gfCNCPoint5[19231] = {X 227.6405, Y 45.0000, Z -7.1667, A 0.000, B 0.000, C 0.000 }
gfCNCPoint5[19232] = {X 227.5362, Y 45.9257, Z -7.1667, A 0.000, B 0.000, C 0.000 }
gfCNCPoint5[19233] = {X 227.2285, Y 46.8050, Z -7.1667, A 0.000, B 0.000, C 0.000 }
gfCNCPoint5[19234] = {X 226.7329, Y 47.5937, Z -7.1667, A 0.000, B 0.000, C 0.000 }
gfCNCPoint5[19235] = {X 226.0742, Y 48.2524, Z -7.1667, A 0.000, B 0.000, C 0.000 }
gfCNCPoint5[19236] = {X 225.2854, Y 48.7480, Z -7.1667, A 0.000, B 0.000, C 0.000 }
gfCNCPoint5[19237] = {X 224.4062, Y 49.0557, Z -7.1667, A 0.000, B 0.000, C 0.000 }
gfCNCPoint5[19238] = {X 223.4805, Y 49.1600, Z -7.1667, A 0.000, B 0.000, C 0.000 }
gfCNCPoint5[19239] = {X 217.0370, Y 49.1600, Z -7.1667, A 0.000, B 0.000, C 0.000 }
gfCNCPoint5[19240] = {X 216.1160, Y 49.0568, Z -7.1667, A 0.000, B 0.000, C 0.000 }
gfCNCPoint5[19241] = {X 215.2406, Y 48.7521, Z -7.1667, A 0.000, B 0.000, C 0.000 }
gfCNCPoint5[19242] = {X 214.4544, Y 48.2613, Z -7.1667, A 0.000, B 0.000, C 0.000 }
gfCNCPoint5[19243] = {X 213.7965, Y 47.6085, Z -7.1667, A 0.000, B 0.000, C 0.000 }
gfCNCPoint5[19244] = {X 213.2993, Y 46.8263, Z -7.1667, A 0.000, B 0.000, C 0.000 }
gfCNCPoint5[19245] = {X 212.9877, Y 45.9534, Z -7.1667, A 0.000, B 0.000, C 0.000 }
gfCNCPoint5[19246] = {X 212.8771, Y 45.0332, Z -7.1667, A 0.000, B 0.000, C 0.000 }
gfCNCPoint5[19247] = {X 212.8770, Y 44.1909, Z -7.1667, A 0.000, B 0.000, C 0.000 }
gfCNCPoint5[19248] = {X 212.9460, Y 43.4438, Z -7.1667, A 0.000, B 0.000, C 0.000 }
gfCNCPoint5[19249] = {X 213.1506, Y 42.7220, Z -7.1667, A 0.000, B 0.000, C 0.000 }
gfCNCPoint5[19250] = {X 213.4838, Y 42.0498, Z -7.1667, A 0.000, B 0.000, C 0.000 }
gfCNCPoint5[19251] = {X 213.9345, Y 41.4500, Z -7.1667, A 0.000, B 0.000, C 0.000 }
gfCNCPoint5[19252] = {X 214.3990, Y 40.9376, Z -7.1667, A 0.000, B 0.000, C 0.000 }
gfCNCPoint5[19253] = {X 214.4039, Y 40.3069, Z -7.1667, A 0.000, B 0.000, C 0.000 }
gfCNCPoint5[19254] = {X 214.4039, Y 28.5737, Z -7.1667, A 0.000, B 0.000, C 0.000 }
gfCNCPoint5[19255] = {X 210.4039, Y 28.5737, Z -7.1667, A 0.000, B 0.000, C 0.000 }
gfCNCPoint5[19256] = {X 214.4839, Y 28.5737, Z -7.1667, A 0.000, B 0.000, C 0.000 }
gfCNCPoint5[19257] = {X 214.4839, Y 17.4614, Z -7.1667, A 0.000, B 0.000, C 0.000 }
gfCNCPoint5[19258] = {X 214.4785, Y 16.7691, Z -7.1667, A 0.000, B 0.000, C 0.000 }
gfCNCPoint5[19259] = {X 214.4828, Y 16.1596, Z -7.1667, A 0.000, B 0.000, C 0.000 }
gfCNCPoint5[19260] = {X 214.4247, Y 16.1121, Z -7.1667, A 0.000, B 0.000, C 0.000 }
gfCNCPoint5[19261] = {X 214.3675, Y 16.0635, Z -7.1667, A 0.000, B 0.000, C 0.000 }
gfCNCPoint5[19262] = {X 213.7773, Y 15.4317, Z -7.1667, A 0.000, B 0.000, C 0.000 }
gfCNCPoint5[19263] = {X 213.3335, Y 14.6898, Z -7.1667, A 0.000, B 0.000, C 0.000 }
gfCNCPoint5[19264] = {X 213.0559, Y 13.8710, Z -7.1667, A 0.000, B 0.000, C 0.000 }
gfCNCPoint5[19265] = {X 212.9572, Y 13.0121, Z -7.1667, A 0.000, B 0.000, C 0.000 }
gfCNCPoint5[19266] = {X 212.9570, Y 12.1868, Z -7.1667, A 0.000, B 0.000, C 0.000 }
gfCNCPoint5[19267] = {X 213.0593, Y 11.2789, Z -7.1667, A 0.000, B 0.000, C 0.000 }
gfCNCPoint5[19268] = {X 213.3611, Y 10.4166, Z -7.1667, A 0.000, B 0.000, C 0.000 }
gfCNCPoint5[19269] = {X 213.8471, Y 9.6430, Z -7.1667, A 0.000, B 0.000, C 0.000 }
gfCNCPoint5[19270] = {X 214.4932, Y 8.9969, Z -7.1667, A 0.000, B 0.000, C 0.000 }
gfCNCPoint5[19271] = {X 215.2668, Y 8.5109, Z -7.1667, A 0.000, B 0.000, C 0.000 }
gfCNCPoint5[19272] = {X 216.1291, Y 8.2091, Z -7.1667, A 0.000, B 0.000, C 0.000 }
gfCNCPoint5[19273] = {X 217.0370, Y 8.1068, Z -7.1667, A 0.000, B 0.000, C 0.000 }
gfCNCPoint5[19274] = {X 223.4805, Y 8.1068, Z -7.1667, A 0.000, B 0.000, C 0.000 }
gfCNCPoint5[19275] = {X 224.3884, Y 8.2091, Z -7.1667, A 0.000, B 0.000, C 0.000 }
gfCNCPoint5[19276] = {X 225.2507, Y 8.5109, Z -7.1667, A 0.000, B 0.000, C 0.000 }
gfCNCPoint5[19277] = {X 226.0243, Y 8.9969, Z -7.1667, A 0.000, B 0.000, C 0.000 }
gfCNCPoint5[19278] = {X 226.6704, Y 9.6430, Z -7.1667, A 0.000, B 0.000, C 0.000 }
gfCNCPoint5[19279] = {X 227.1564, Y 10.4166, Z -7.1667, A 0.000, B 0.000, C 0.000 }
gfCNCPoint5[19280] = {X 227.4582, Y 11.2789, Z -7.1667, A 0.000, B 0.000, C 0.000 }
gfCNCPoint5[19281] = {X 227.5605, Y 12.1868, Z -7.1667, A 0.000, B 0.000, C 0.000 }
gfCNCPoint5[19282] = {X 227.5605, Y 12.9782, Z -7.1667, A 0.000, B 0.000, C 0.000 }
gfCNCPoint5[19283] = {X 227.4589, Y 13.8829, Z -7.1667, A 0.000, B 0.000, C 0.000 }
gfCNCPoint5[19284] = {X 227.1591, Y 14.7427, Z -7.1667, A 0.000, B 0.000, C 0.000 }
gfCNCPoint5[19285] = {X 226.6762, Y 15.5145, Z -7.1667, A 0.000, B 0.000, C 0.000 }
gfCNCPoint5[19286] = {X 226.0341, Y 16.1600, Z -7.1667, A 0.000, B 0.000, C 0.000 }
gfCNCPoint5[19287] = {X 226.0351, Y 41.0283, Z -7.1667, A 0.000, B 0.000, C 0.000 }
gfCNCPoint5[19288] = {X 226.1412, Y 41.1157, Z -7.1667, A 0.000, B 0.000, C 0.000 }
gfCNCPoint5[19289] = {X 226.7344, Y 41.7474, Z -7.1667, A 0.000, B 0.000, C 0.000 }
gfCNCPoint5[19290] = {X 227.1808, Y 42.4901, Z -7.1667, A 0.000, B 0.000, C 0.000 }
gfCNCPoint5[19291] = {X 227.4603, Y 43.3104, Z -7.1667, A 0.000, B 0.000, C 0.000 }
gfCNCPoint5[19292] = {X 227.5603, Y 44.1712, Z -7.1667, A 0.000, B 0.000, C 0.000 }
gfCNCPoint5[19293] = {X 227.5605, Y 45.0000, Z -7.1667, A 0.000, B 0.000, C 0.000 }
gfCNCPoint5[19294] = {X 227.4582, Y 45.9079, Z -7.1667, A 0.000, B 0.000, C 0.000 }
gfCNCPoint5[19295] = {X 227.1564, Y 46.7702, Z -7.1667, A 0.000, B 0.000, C 0.000 }
gfCNCPoint5[19296] = {X 226.6704, Y 47.5438, Z -7.1667, A 0.000, B 0.000, C 0.000 }
gfCNCPoint5[19297] = {X 226.0243, Y 48.1899, Z -7.1667, A 0.000, B 0.000, C 0.000 }
gfCNCPoint5[19298] = {X 225.2507, Y 48.6760, Z -7.1667, A 0.000, B 0.000, C 0.000 }
gfCNCPoint5[19299] = {X 224.3884, Y 48.9777, Z -7.1667, A 0.000, B 0.000, C 0.000 }
gfCNCPoint5[19300] = {X 223.4805, Y 49.0800, Z -7.1667, A 0.000, B 0.000, C 0.000 }
gfCNCPoint5[19301] = {X 217.0370, Y 49.0800, Z -7.1667, A 0.000, B 0.000, C 0.000 }
gfCNCPoint5[19302] = {X 216.1337, Y 48.9787, Z -7.1667, A 0.000, B 0.000, C 0.000 }
gfCNCPoint5[19303] = {X 215.2752, Y 48.6800, Z -7.1667, A 0.000, B 0.000, C 0.000 }
gfCNCPoint5[19304] = {X 214.5041, Y 48.1986, Z -7.1667, A 0.000, B 0.000, C 0.000 }
gfCNCPoint5[19305] = {X 213.8588, Y 47.5584, Z -7.1667, A 0.000, B 0.000, C 0.000 }
gfCNCPoint5[19306] = {X 213.3712, Y 46.7912, Z -7.1667, A 0.000, B 0.000, C 0.000 }
gfCNCPoint5[19307] = {X 213.0656, Y 45.9351, Z -7.1667, A 0.000, B 0.000, C 0.000 }
gfCNCPoint5[19308] = {X 212.9571, Y 45.0325, Z -7.1667, A 0.000, B 0.000, C 0.000 }
gfCNCPoint5[19309] = {X 212.9570, Y 44.1909, Z -7.1667, A 0.000, B 0.000, C 0.000 }
gfCNCPoint5[19310] = {X 213.0246, Y 43.4585, Z -7.1667, A 0.000, B 0.000, C 0.000 }
gfCNCPoint5[19311] = {X 213.2252, Y 42.7508, Z -7.1667, A 0.000, B 0.000, C 0.000 }
gfCNCPoint5[19312] = {X 213.5519, Y 42.0918, Z -7.1667, A 0.000, B 0.000, C 0.000 }
gfCNCPoint5[19313] = {X 213.9938, Y 41.5037, Z -7.1667, A 0.000, B 0.000, C 0.000 }
gfCNCPoint5[19314] = {X 214.4788, Y 40.9687, Z -7.1667, A 0.000, B 0.000, C 0.000 }
gfCNCPoint5[19315] = {X 214.4839, Y 40.3072, Z -7.1667, A 0.000, B 0.000, C 0.000 }
gfCNCPoint5[19316] = {X 214.4839, Y 28.5737, Z -7.1667, A 0.000, B 0.000, C 0.000 }
gfCNCPoint5[19317] = {X 210.4839, Y 28.5737, Z -7.1667, A 0.000, B 0.000, C 0.000 }
gfCNCPoint5[19318] = {X 214.5639, Y 28.5737, Z -7.1667, A 0.000, B 0.000, C 0.000 }
gfCNCPoint5[19319] = {X 214.5639, Y 17.4611, Z -7.1667, A 0.000, B 0.000, C 0.000 }
gfCNCPoint5[19320] = {X 214.5585, Y 16.7687, Z -7.1667, A 0.000, B 0.000, C 0.000 }
gfCNCPoint5[19321] = {X 214.5580, Y 16.1871, Z -7.1667, A 0.000, B 0.000, C 0.000 }
gfCNCPoint5[19322] = {X 214.5756, Y 16.1310, Z -7.1667, A 0.000, B 0.000, C 0.000 }
gfCNCPoint5[19323] = {X 214.4969, Y 16.0680, Z -7.1667, A 0.000, B 0.000, C 0.000 }
gfCNCPoint5[19324] = {X 214.4199, Y 16.0030, Z -7.1667, A 0.000, B 0.000, C 0.000 }
gfCNCPoint5[19325] = {X 213.8362, Y 15.3769, Z -7.1667, A 0.000, B 0.000, C 0.000 }
gfCNCPoint5[19326] = {X 213.3991, Y 14.6410, Z -7.1667, A 0.000, B 0.000, C 0.000 }
gfCNCPoint5[19327] = {X 213.1286, Y 13.8290, Z -7.1667, A 0.000, B 0.000, C 0.000 }
gfCNCPoint5[19328] = {X 213.0370, Y 12.9780, Z -7.1667, A 0.000, B 0.000, C 0.000 }
gfCNCPoint5[19329] = {X 213.0370, Y 12.1868, Z -7.1667, A 0.000, B 0.000, C 0.000 }
gfCNCPoint5[19330] = {X 213.1373, Y 11.2967, Z -7.1667, A 0.000, B 0.000, C 0.000 }
gfCNCPoint5[19331] = {X 213.4331, Y 10.4513, Z -7.1667, A 0.000, B 0.000, C 0.000 }
gfCNCPoint5[19332] = {X 213.9097, Y 9.6929, Z -7.1667, A 0.000, B 0.000, C 0.000 }
gfCNCPoint5[19333] = {X 214.5431, Y 9.0595, Z -7.1667, A 0.000, B 0.000, C 0.000 }
gfCNCPoint5[19334] = {X 215.3015, Y 8.5829, Z -7.1667, A 0.000, B 0.000, C 0.000 }
gfCNCPoint5[19335] = {X 216.1469, Y 8.2871, Z -7.1667, A 0.000, B 0.000, C 0.000 }
gfCNCPoint5[19336] = {X 217.0370, Y 8.1868, Z -7.1667, A 0.000, B 0.000, C 0.000 }
gfCNCPoint5[19337] = {X 223.4805, Y 8.1868, Z -7.1667, A 0.000, B 0.000, C 0.000 }
gfCNCPoint5[19338] = {X 224.3706, Y 8.2871, Z -7.1667, A 0.000, B 0.000, C 0.000 }
gfCNCPoint5[19339] = {X 225.2160, Y 8.5829, Z -7.1667, A 0.000, B 0.000, C 0.000 }
gfCNCPoint5[19340] = {X 225.9744, Y 9.0595, Z -7.1667, A 0.000, B 0.000, C 0.000 }
gfCNCPoint5[19341] = {X 226.6078, Y 9.6929, Z -7.1667, A 0.000, B 0.000, C 0.000 }
gfCNCPoint5[19342] = {X 227.0844, Y 10.4513, Z -7.1667, A 0.000, B 0.000, C 0.000 }
gfCNCPoint5[19343] = {X 227.3802, Y 11.2967, Z -7.1667, A 0.000, B 0.000, C 0.000 }
gfCNCPoint5[19344] = {X 227.4805, Y 12.1868, Z -7.1667, A 0.000, B 0.000, C 0.000 }
gfCNCPoint5[19345] = {X 227.4803, Y 13.0192, Z -7.1667, A 0.000, B 0.000, C 0.000 }
gfCNCPoint5[19346] = {X 227.3717, Y 13.9045, Z -7.1667, A 0.000, B 0.000, C 0.000 }
gfCNCPoint5[19347] = {X 227.0697, Y 14.7437, Z -7.1667, A 0.000, B 0.000, C 0.000 }
gfCNCPoint5[19348] = {X 226.5892, Y 15.4951, Z -7.1667, A 0.000, B 0.000, C 0.000 }
gfCNCPoint5[19349] = {X 225.9541, Y 16.1214, Z -7.1667, A 0.000, B 0.000, C 0.000 }
gfCNCPoint5[19350] = {X 225.9551, Y 41.0660, Z -7.1667, A 0.000, B 0.000, C 0.000 }
gfCNCPoint5[19351] = {X 226.0938, Y 41.1805, Z -7.1667, A 0.000, B 0.000, C 0.000 }
gfCNCPoint5[19352] = {X 226.6790, Y 41.8068, Z -7.1667, A 0.000, B 0.000, C 0.000 }
gfCNCPoint5[19353] = {X 227.1173, Y 42.5435, Z -7.1667, A 0.000, B 0.000, C 0.000 }
gfCNCPoint5[19354] = {X 227.3886, Y 43.3566, Z -7.1667, A 0.000, B 0.000, C 0.000 }
gfCNCPoint5[19355] = {X 227.4805, Y 44.2089, Z -7.1667, A 0.000, B 0.000, C 0.000 }
gfCNCPoint5[19356] = {X 227.4805, Y 45.0000, Z -7.1667, A 0.000, B 0.000, C 0.000 }
gfCNCPoint5[19357] = {X 227.3802, Y 45.8901, Z -7.1667, A 0.000, B 0.000, C 0.000 }
gfCNCPoint5[19358] = {X 227.0844, Y 46.7355, Z -7.1667, A 0.000, B 0.000, C 0.000 }
gfCNCPoint5[19359] = {X 226.6078, Y 47.4940, Z -7.1667, A 0.000, B 0.000, C 0.000 }
gfCNCPoint5[19360] = {X 225.9744, Y 48.1273, Z -7.1667, A 0.000, B 0.000, C 0.000 }
gfCNCPoint5[19361] = {X 225.2160, Y 48.6039, Z -7.1667, A 0.000, B 0.000, C 0.000 }
gfCNCPoint5[19362] = {X 224.3706, Y 48.8997, Z -7.1667, A 0.000, B 0.000, C 0.000 }
gfCNCPoint5[19363] = {X 223.4805, Y 49.0000, Z -7.1667, A 0.000, B 0.000, C 0.000 }
gfCNCPoint5[19364] = {X 217.0370, Y 49.0000, Z -7.1667, A 0.000, B 0.000, C 0.000 }
gfCNCPoint5[19365] = {X 216.1469, Y 48.8997, Z -7.1667, A 0.000, B 0.000, C 0.000 }
gfCNCPoint5[19366] = {X 215.3015, Y 48.6039, Z -7.1667, A 0.000, B 0.000, C 0.000 }
gfCNCPoint5[19367] = {X 214.5430, Y 48.1273, Z -7.1667, A 0.000, B 0.000, C 0.000 }
gfCNCPoint5[19368] = {X 213.9097, Y 47.4939, Z -7.1667, A 0.000, B 0.000, C 0.000 }
gfCNCPoint5[19369] = {X 213.4331, Y 46.7355, Z -7.1667, A 0.000, B 0.000, C 0.000 }
gfCNCPoint5[19370] = {X 213.1373, Y 45.8901, Z -7.1667, A 0.000, B 0.000, C 0.000 }
gfCNCPoint5[19371] = {X 213.0370, Y 45.0000, Z -7.1667, A 0.000, B 0.000, C 0.000 }
gfCNCPoint5[19372] = {X 213.0370, Y 44.1909, Z -7.1667, A 0.000, B 0.000, C 0.000 }
gfCNCPoint5[19373] = {X 213.1546, Y 43.2380, Z -7.1667, A 0.000, B 0.000, C 0.000 }
gfCNCPoint5[19374] = {X 213.5002, Y 42.3423, Z -7.1667, A 0.000, B 0.000, C 0.000 }
gfCNCPoint5[19375] = {X 214.0531, Y 41.5574, Z -7.1667, A 0.000, B 0.000, C 0.000 }
gfCNCPoint5[19376] = {X 214.5585, Y 40.9999, Z -7.1667, A 0.000, B 0.000, C 0.000 }
gfCNCPoint5[19377] = {X 214.5639, Y 40.3075, Z -7.1667, A 0.000, B 0.000, C 0.000 }
gfCNCPoint5[19378] = {X 214.5639, Y 28.5737, Z -7.1667, A 0.000, B 0.000, C 0.000 }
gfCNCPoint5[19379] = {X 210.4839, Y 28.5737, Z -7.1667, A 0.000, B 0.000, C 0.000 }
gfCNCPoint5[19380] = {X 210.4839, Y 28.5737, Z -4.1667, A 0.000, B 0.000, C 0.000 }
gfCNCPoint5[19381] = {X 210.4839, Y 28.5737, Z 11.0000, A 0.000, B 0.000, C 0.000 }
gfCNCPoint5[19382] = {X 273.6047, Y 28.5936, Z 11.0000, A 0.000, B 0.000, C 0.000 }
gfCNCPoint5[19383] = {X 273.6047, Y 28.5936, Z -4.1667, A 0.000, B 0.000, C 0.000 }
gfCNCPoint5[19384] = {X 273.6047, Y 28.5936, Z -7.1667, A 0.000, B 0.000, C 0.000 }
gfCNCPoint5[19385] = {X 269.5247, Y 28.5937, Z -7.1667, A 0.000, B 0.000, C 0.000 }
gfCNCPoint5[19386] = {X 269.5248, Y 40.9141, Z -7.1667, A 0.000, B 0.000, C 0.000 }
gfCNCPoint5[19387] = {X 269.5381, Y 40.9251, Z -7.1667, A 0.000, B 0.000, C 0.000 }
gfCNCPoint5[19388] = {X 270.1703, Y 41.5946, Z -7.1667, A 0.000, B 0.000, C 0.000 }
gfCNCPoint5[19389] = {X 270.6462, Y 42.3828, Z -7.1667, A 0.000, B 0.000, C 0.000 }
gfCNCPoint5[19390] = {X 270.9442, Y 43.2540, Z -7.1667, A 0.000, B 0.000, C 0.000 }
gfCNCPoint5[19391] = {X 271.0508, Y 44.1686, Z -7.1667, A 0.000, B 0.000, C 0.000 }
gfCNCPoint5[19392] = {X 271.0510, Y 45.0000, Z -7.1667, A 0.000, B 0.000, C 0.000 }
gfCNCPoint5[19393] = {X 270.9427, Y 45.9613, Z -7.1667, A 0.000, B 0.000, C 0.000 }
gfCNCPoint5[19394] = {X 270.6232, Y 46.8744, Z -7.1667, A 0.000, B 0.000, C 0.000 }
gfCNCPoint5[19395] = {X 270.1085, Y 47.6935, Z -7.1667, A 0.000, B 0.000, C 0.000 }
gfCNCPoint5[19396] = {X 269.4245, Y 48.3775, Z -7.1667, A 0.000, B 0.000, C 0.000 }
gfCNCPoint5[19397] = {X 268.6054, Y 48.8922, Z -7.1667, A 0.000, B 0.000, C 0.000 }
gfCNCPoint5[19398] = {X 267.6923, Y 49.2117, Z -7.1667, A 0.000, B 0.000, C 0.000 }
gfCNCPoint5[19399] = {X 266.7310, Y 49.3200, Z -7.1667, A 0.000, B 0.000, C 0.000 }
gfCNCPoint5[19400] = {X 260.2876, Y 49.3200, Z -7.1667, A 0.000, B 0.000, C 0.000 }
gfCNCPoint5[19401] = {X 259.3310, Y 49.2128, Z -7.1667, A 0.000, B 0.000, C 0.000 }
gfCNCPoint5[19402] = {X 258.4219, Y 48.8963, Z -7.1667, A 0.000, B 0.000, C 0.000 }
gfCNCPoint5[19403] = {X 257.6054, Y 48.3865, Z -7.1667, A 0.000, B 0.000, C 0.000 }
gfCNCPoint5[19404] = {X 256.9221, Y 47.7085, Z -7.1667, A 0.000, B 0.000, C 0.000 }
gfCNCPoint5[19405] = {X 256.4059, Y 46.8960, Z -7.1667, A 0.000, B 0.000, C 0.000 }
gfCNCPoint5[19406] = {X 256.0824, Y 45.9894, Z -7.1667, A 0.000, B 0.000, C 0.000 }
gfCNCPoint5[19407] = {X 255.9677, Y 45.0336, Z -7.1667, A 0.000, B 0.000, C 0.000 }
gfCNCPoint5[19408] = {X 255.9680, Y 44.1494, Z -7.1667, A 0.000, B 0.000, C 0.000 }
gfCNCPoint5[19409] = {X 256.0784, Y 43.2364, Z -7.1667, A 0.000, B 0.000, C 0.000 }
gfCNCPoint5[19410] = {X 256.3796, Y 42.3675, Z -7.1667, A 0.000, B 0.000, C 0.000 }
gfCNCPoint5[19411] = {X 256.8579, Y 41.5821, Z -7.1667, A 0.000, B 0.000, C 0.000 }
gfCNCPoint5[19412] = {X 257.4915, Y 40.9157, Z -7.1667, A 0.000, B 0.000, C 0.000 }
gfCNCPoint5[19413] = {X 257.4915, Y 34.4738, Z -7.1667, A 0.000, B 0.000, C 0.000 }
gfCNCPoint5[19414] = {X 254.7687, Y 34.4738, Z -7.1667, A 0.000, B 0.000, C 0.000 }
gfCNCPoint5[19415] = {X 250.4840, Y 42.8193, Z -7.1667, A 0.000, B 0.000, C 0.000 }
gfCNCPoint5[19416] = {X 250.6528, Y 43.4866, Z -7.1667, A 0.000, B 0.000, C 0.000 }
gfCNCPoint5[19417] = {X 250.7134, Y 44.1723, Z -7.1667, A 0.000, B 0.000, C 0.000 }
gfCNCPoint5[19418] = {X 250.7136, Y 45.0000, Z -7.1667, A 0.000, B 0.000, C 0.000 }
gfCNCPoint5[19419] = {X 250.6052, Y 45.9613, Z -7.1667, A 0.000, B 0.000, C 0.000 }
gfCNCPoint5[19420] = {X 250.2857, Y 46.8744, Z -7.1667, A 0.000, B 0.000, C 0.000 }
gfCNCPoint5[19421] = {X 249.7711, Y 47.6935, Z -7.1667, A 0.000, B 0.000, C 0.000 }
gfCNCPoint5[19422] = {X 249.0870, Y 48.3775, Z -7.1667, A 0.000, B 0.000, C 0.000 }
gfCNCPoint5[19423] = {X 248.2679, Y 48.8922, Z -7.1667, A 0.000, B 0.000, C 0.000 }
gfCNCPoint5[19424] = {X 247.3548, Y 49.2117, Z -7.1667, A 0.000, B 0.000, C 0.000 }
gfCNCPoint5[19425] = {X 246.3936, Y 49.3200, Z -7.1667, A 0.000, B 0.000, C 0.000 }
gfCNCPoint5[19426] = {X 239.8075, Y 49.3200, Z -7.1667, A 0.000, B 0.000, C 0.000 }
gfCNCPoint5[19427] = {X 238.8462, Y 49.2117, Z -7.1667, A 0.000, B 0.000, C 0.000 }
gfCNCPoint5[19428] = {X 237.9332, Y 48.8922, Z -7.1667, A 0.000, B 0.000, C 0.000 }
gfCNCPoint5[19429] = {X 237.1141, Y 48.3775, Z -7.1667, A 0.000, B 0.000, C 0.000 }
gfCNCPoint5[19430] = {X 236.4300, Y 47.6935, Z -7.1667, A 0.000, B 0.000, C 0.000 }
gfCNCPoint5[19431] = {X 235.9153, Y 46.8745, Z -7.1667, A 0.000, B 0.000, C 0.000 }
gfCNCPoint5[19432] = {X 235.5958, Y 45.9614, Z -7.1667, A 0.000, B 0.000, C 0.000 }
gfCNCPoint5[19433] = {X 235.4875, Y 45.0001, Z -7.1667, A 0.000, B 0.000, C 0.000 }
gfCNCPoint5[19434] = {X 235.4879, Y 44.1494, Z -7.1667, A 0.000, B 0.000, C 0.000 }
gfCNCPoint5[19435] = {X 235.5856, Y 43.2935, Z -7.1667, A 0.000, B 0.000, C 0.000 }
gfCNCPoint5[19436] = {X 235.8511, Y 42.4740, Z -7.1667, A 0.000, B 0.000, C 0.000 }
gfCNCPoint5[19437] = {X 236.2739, Y 41.7236, Z -7.1667, A 0.000, B 0.000, C 0.000 }
gfCNCPoint5[19438] = {X 236.8373, Y 41.0719, Z -7.1667, A 0.000, B 0.000, C 0.000 }
gfCNCPoint5[19439] = {X 237.5187, Y 40.5449, Z -7.1667, A 0.000, B 0.000, C 0.000 }
gfCNCPoint5[19440] = {X 238.2911, Y 40.1637, Z -7.1667, A 0.000, B 0.000, C 0.000 }
gfCNCPoint5[19441] = {X 242.2799, Y 32.3561, Z -7.1667, A 0.000, B 0.000, C 0.000 }
gfCNCPoint5[19442] = {X 241.1098, Y 31.5695, Z -7.1667, A 0.000, B 0.000, C 0.000 }
gfCNCPoint5[19443] = {X 240.0466, Y 30.6436, Z -7.1667, A 0.000, B 0.000, C 0.000 }
gfCNCPoint5[19444] = {X 239.1067, Y 29.5928, Z -7.1667, A 0.000, B 0.000, C 0.000 }
gfCNCPoint5[19445] = {X 238.3046, Y 28.4332, Z -7.1667, A 0.000, B 0.000, C 0.000 }
gfCNCPoint5[19446] = {X 237.6529, Y 27.1830, Z -7.1667, A 0.000, B 0.000, C 0.000 }
gfCNCPoint5[19447] = {X 237.1616, Y 25.8615, Z -7.1667, A 0.000, B 0.000, C 0.000 }
gfCNCPoint5[19448] = {X 236.7414, Y 24.0500, Z -7.1667, A 0.000, B 0.000, C 0.000 }
gfCNCPoint5[19449] = {X 236.5273, Y 22.2028, Z -7.1667, A 0.000, B 0.000, C 0.000 }
gfCNCPoint5[19450] = {X 236.5220, Y 20.3432, Z -7.1667, A 0.000, B 0.000, C 0.000 }
gfCNCPoint5[19451] = {X 236.7254, Y 18.4948, Z -7.1667, A 0.000, B 0.000, C 0.000 }
gfCNCPoint5[19452] = {X 237.1352, Y 16.6809, Z -7.1667, A 0.000, B 0.000, C 0.000 }
gfCNCPoint5[19453] = {X 237.7057, Y 15.1051, Z -7.1667, A 0.000, B 0.000, C 0.000 }
gfCNCPoint5[19454] = {X 238.4928, Y 13.6255, Z -7.1667, A 0.000, B 0.000, C 0.000 }
gfCNCPoint5[19455] = {X 239.4808, Y 12.2718, Z -7.1667, A 0.000, B 0.000, C 0.000 }
gfCNCPoint5[19456] = {X 240.6498, Y 11.0710, Z -7.1667, A 0.000, B 0.000, C 0.000 }
gfCNCPoint5[19457] = {X 241.9766, Y 10.0471, Z -7.1667, A 0.000, B 0.000, C 0.000 }
gfCNCPoint5[19458] = {X 243.4345, Y 9.2206, Z -7.1667, A 0.000, B 0.000, C 0.000 }
gfCNCPoint5[19459] = {X 244.9944, Y 8.6080, Z -7.1667, A 0.000, B 0.000, C 0.000 }
gfCNCPoint5[19460] = {X 246.6252, Y 8.2216, Z -7.1667, A 0.000, B 0.000, C 0.000 }
gfCNCPoint5[19461] = {X 248.7221, Y 7.9501, Z -7.1667, A 0.000, B 0.000, C 0.000 }
gfCNCPoint5[19462] = {X 250.8350, Y 7.8696, Z -7.1667, A 0.000, B 0.000, C 0.000 }
gfCNCPoint5[19463] = {X 266.7633, Y 7.8696, Z -7.1667, A 0.000, B 0.000, C 0.000 }
gfCNCPoint5[19464] = {X 267.7187, Y 7.9843, Z -7.1667, A 0.000, B 0.000, C 0.000 }
gfCNCPoint5[19465] = {X 268.6250, Y 8.3076, Z -7.1667, A 0.000, B 0.000, C 0.000 }
gfCNCPoint5[19466] = {X 269.4373, Y 8.8234, Z -7.1667, A 0.000, B 0.000, C 0.000 }
gfCNCPoint5[19467] = {X 270.1154, Y 9.5061, Z -7.1667, A 0.000, B 0.000, C 0.000 }
gfCNCPoint5[19468] = {X 270.6256, Y 10.3219, Z -7.1667, A 0.000, B 0.000, C 0.000 }
gfCNCPoint5[19469] = {X 270.9427, Y 11.2303, Z -7.1667, A 0.000, B 0.000, C 0.000 }
gfCNCPoint5[19470] = {X 271.0510, Y 12.1865, Z -7.1667, A 0.000, B 0.000, C 0.000 }
gfCNCPoint5[19471] = {X 271.0508, Y 13.0225, Z -7.1667, A 0.000, B 0.000, C 0.000 }
gfCNCPoint5[19472] = {X 270.9425, Y 13.9402, Z -7.1667, A 0.000, B 0.000, C 0.000 }
gfCNCPoint5[19473] = {X 270.6415, Y 14.8139, Z -7.1667, A 0.000, B 0.000, C 0.000 }
gfCNCPoint5[19474] = {X 270.1616, Y 15.6036, Z -7.1667, A 0.000, B 0.000, C 0.000 }
gfCNCPoint5[19475] = {X 269.5247, Y 16.2732, Z -7.1667, A 0.000, B 0.000, C 0.000 }
gfCNCPoint5[19476] = {X 269.5247, Y 28.5937, Z -7.1667, A 0.000, B 0.000, C 0.000 }
gfCNCPoint5[19477] = {X 273.5247, Y 28.5936, Z -7.1667, A 0.000, B 0.000, C 0.000 }
gfCNCPoint5[19478] = {X 269.4447, Y 28.5937, Z -7.1667, A 0.000, B 0.000, C 0.000 }
gfCNCPoint5[19479] = {X 269.4448, Y 40.9519, Z -7.1667, A 0.000, B 0.000, C 0.000 }
gfCNCPoint5[19480] = {X 269.4867, Y 40.9864, Z -7.1667, A 0.000, B 0.000, C 0.000 }
gfCNCPoint5[19481] = {X 270.1069, Y 41.6434, Z -7.1667, A 0.000, B 0.000, C 0.000 }
gfCNCPoint5[19482] = {X 270.5738, Y 42.4170, Z -7.1667, A 0.000, B 0.000, C 0.000 }
gfCNCPoint5[19483] = {X 270.8662, Y 43.2719, Z -7.1667, A 0.000, B 0.000, C 0.000 }
gfCNCPoint5[19484] = {X 270.9708, Y 44.1693, Z -7.1667, A 0.000, B 0.000, C 0.000 }
gfCNCPoint5[19485] = {X 270.9710, Y 45.0000, Z -7.1667, A 0.000, B 0.000, C 0.000 }
gfCNCPoint5[19486] = {X 270.8647, Y 45.9435, Z -7.1667, A 0.000, B 0.000, C 0.000 }
gfCNCPoint5[19487] = {X 270.5511, Y 46.8397, Z -7.1667, A 0.000, B 0.000, C 0.000 }
gfCNCPoint5[19488] = {X 270.0460, Y 47.6436, Z -7.1667, A 0.000, B 0.000, C 0.000 }
gfCNCPoint5[19489] = {X 269.3746, Y 48.3150, Z -7.1667, A 0.000, B 0.000, C 0.000 }
gfCNCPoint5[19490] = {X 268.5707, Y 48.8201, Z -7.1667, A 0.000, B 0.000, C 0.000 }
gfCNCPoint5[19491] = {X 267.6745, Y 49.1337, Z -7.1667, A 0.000, B 0.000, C 0.000 }
gfCNCPoint5[19492] = {X 266.7310, Y 49.2400, Z -7.1667, A 0.000, B 0.000, C 0.000 }
gfCNCPoint5[19493] = {X 260.2876, Y 49.2400, Z -7.1667, A 0.000, B 0.000, C 0.000 }
gfCNCPoint5[19494] = {X 259.3487, Y 49.1347, Z -7.1667, A 0.000, B 0.000, C 0.000 }
gfCNCPoint5[19495] = {X 258.4564, Y 48.8242, Z -7.1667, A 0.000, B 0.000, C 0.000 }
gfCNCPoint5[19496] = {X 257.6550, Y 48.3238, Z -7.1667, A 0.000, B 0.000, C 0.000 }
gfCNCPoint5[19497] = {X 256.9844, Y 47.6583, Z -7.1667, A 0.000, B 0.000, C 0.000 }
gfCNCPoint5[19498] = {X 256.4777, Y 46.8609, Z -7.1667, A 0.000, B 0.000, C 0.000 }
gfCNCPoint5[19499] = {X 256.1603, Y 45.9711, Z -7.1667, A 0.000, B 0.000, C 0.000 }
gfCNCPoint5[19500] = {X 256.0477, Y 45.0330, Z -7.1667, A 0.000, B 0.000, C 0.000 }
gfCNCPoint5[19501] = {X 256.0480, Y 44.1505, Z -7.1667, A 0.000, B 0.000, C 0.000 }
gfCNCPoint5[19502] = {X 256.1585, Y 43.2454, Z -7.1667, A 0.000, B 0.000, C 0.000 }
gfCNCPoint5[19503] = {X 256.4599, Y 42.3850, Z -7.1667, A 0.000, B 0.000, C 0.000 }
gfCNCPoint5[19504] = {X 256.9383, Y 41.6088, Z -7.1667, A 0.000, B 0.000, C 0.000 }
gfCNCPoint5[19505] = {X 257.5715, Y 40.9529, Z -7.1667, A 0.000, B 0.000, C 0.000 }
gfCNCPoint5[19506] = {X 257.5715, Y 34.3938, Z -7.1667, A 0.000, B 0.000, C 0.000 }
gfCNCPoint5[19507] = {X 254.7198, Y 34.3938, Z -7.1667, A 0.000, B 0.000, C 0.000 }
gfCNCPoint5[19508] = {X 250.3972, Y 42.8130, Z -7.1667, A 0.000, B 0.000, C 0.000 }
gfCNCPoint5[19509] = {X 250.5710, Y 43.4833, Z -7.1667, A 0.000, B 0.000, C 0.000 }
gfCNCPoint5[19510] = {X 250.6334, Y 44.1730, Z -7.1667, A 0.000, B 0.000, C 0.000 }
gfCNCPoint5[19511] = {X 250.6336, Y 45.0000, Z -7.1667, A 0.000, B 0.000, C 0.000 }
gfCNCPoint5[19512] = {X 250.5273, Y 45.9435, Z -7.1667, A 0.000, B 0.000, C 0.000 }
gfCNCPoint5[19513] = {X 250.2137, Y 46.8397, Z -7.1667, A 0.000, B 0.000, C 0.000 }
gfCNCPoint5[19514] = {X 249.7085, Y 47.6436, Z -7.1667, A 0.000, B 0.000, C 0.000 }
gfCNCPoint5[19515] = {X 249.0372, Y 48.3150, Z -7.1667, A 0.000, B 0.000, C 0.000 }
gfCNCPoint5[19516] = {X 248.2332, Y 48.8201, Z -7.1667, A 0.000, B 0.000, C 0.000 }
gfCNCPoint5[19517] = {X 247.3370, Y 49.1337, Z -7.1667, A 0.000, B 0.000, C 0.000 }
gfCNCPoint5[19518] = {X 246.3936, Y 49.2400, Z -7.1667, A 0.000, B 0.000, C 0.000 }
gfCNCPoint5[19519] = {X 239.8075, Y 49.2400, Z -7.1667, A 0.000, B 0.000, C 0.000 }
gfCNCPoint5[19520] = {X 238.8640, Y 49.1337, Z -7.1667, A 0.000, B 0.000, C 0.000 }
gfCNCPoint5[19521] = {X 237.9679, Y 48.8201, Z -7.1667, A 0.000, B 0.000, C 0.000 }
gfCNCPoint5[19522] = {X 237.1639, Y 48.3150, Z -7.1667, A 0.000, B 0.000, C 0.000 }
gfCNCPoint5[19523] = {X 236.4926, Y 47.6436, Z -7.1667, A 0.000, B 0.000, C 0.000 }
gfCNCPoint5[19524] = {X 235.9874, Y 46.8397, Z -7.1667, A 0.000, B 0.000, C 0.000 }
gfCNCPoint5[19525] = {X 235.6738, Y 45.9436, Z -7.1667, A 0.000, B 0.000, C 0.000 }
gfCNCPoint5[19526] = {X 235.5675, Y 45.0001, Z -7.1667, A 0.000, B 0.000, C 0.000 }
gfCNCPoint5[19527] = {X 235.5679, Y 44.1505, Z -7.1667, A 0.000, B 0.000, C 0.000 }
gfCNCPoint5[19528] = {X 235.6649, Y 43.3054, Z -7.1667, A 0.000, B 0.000, C 0.000 }
gfCNCPoint5[19529] = {X 235.9285, Y 42.4967, Z -7.1667, A 0.000, B 0.000, C 0.000 }
gfCNCPoint5[19530] = {X 236.3483, Y 41.7570, Z -7.1667, A 0.000, B 0.000, C 0.000 }
gfCNCPoint5[19531] = {X 236.9073, Y 41.1158, Z -7.1667, A 0.000, B 0.000, C 0.000 }
gfCNCPoint5[19532] = {X 237.5830, Y 40.5992, Z -7.1667, A 0.000, B 0.000, C 0.000 }
gfCNCPoint5[19533] = {X 238.3482, Y 40.2278, Z -7.1667, A 0.000, B 0.000, C 0.000 }
gfCNCPoint5[19534] = {X 242.3856, Y 32.3250, Z -7.1667, A 0.000, B 0.000, C 0.000 }
gfCNCPoint5[19535] = {X 241.2086, Y 31.5442, Z -7.1667, A 0.000, B 0.000, C 0.000 }
gfCNCPoint5[19536] = {X 240.1387, Y 30.6220, Z -7.1667, A 0.000, B 0.000, C 0.000 }
gfCNCPoint5[19537] = {X 239.1929, Y 29.5729, Z -7.1667, A 0.000, B 0.000, C 0.000 }
gfCNCPoint5[19538] = {X 238.3862, Y 28.4134, Z -7.1667, A 0.000, B 0.000, C 0.000 }
gfCNCPoint5[19539] = {X 237.7311, Y 27.1620, Z -7.1667, A 0.000, B 0.000, C 0.000 }
gfCNCPoint5[19540] = {X 237.2382, Y 25.8383, Z -7.1667, A 0.000, B 0.000, C 0.000 }
gfCNCPoint5[19541] = {X 236.8201, Y 24.0357, Z -7.1667, A 0.000, B 0.000, C 0.000 }
gfCNCPoint5[19542] = {X 236.6071, Y 22.1976, Z -7.1667, A 0.000, B 0.000, C 0.000 }
gfCNCPoint5[19543] = {X 236.6019, Y 20.3472, Z -7.1667, A 0.000, B 0.000, C 0.000 }
gfCNCPoint5[19544] = {X 236.8044, Y 18.5078, Z -7.1667, A 0.000, B 0.000, C 0.000 }
gfCNCPoint5[19545] = {X 237.2121, Y 16.7029, Z -7.1667, A 0.000, B 0.000, C 0.000 }
gfCNCPoint5[19546] = {X 237.7788, Y 15.1376, Z -7.1667, A 0.000, B 0.000, C 0.000 }
gfCNCPoint5[19547] = {X 238.5606, Y 13.6680, Z -7.1667, A 0.000, B 0.000, C 0.000 }
gfCNCPoint5[19548] = {X 239.5420, Y 12.3233, Z -7.1667, A 0.000, B 0.000, C 0.000 }
gfCNCPoint5[19549] = {X 240.7032, Y 11.1306, Z -7.1667, A 0.000, B 0.000, C 0.000 }
gfCNCPoint5[19550] = {X 242.0211, Y 10.1135, Z -7.1667, A 0.000, B 0.000, C 0.000 }
gfCNCPoint5[19551] = {X 243.4692, Y 9.2926, Z -7.1667, A 0.000, B 0.000, C 0.000 }
gfCNCPoint5[19552] = {X 245.0187, Y 8.6842, Z -7.1667, A 0.000, B 0.000, C 0.000 }
gfCNCPoint5[19553] = {X 246.6386, Y 8.3005, Z -7.1667, A 0.000, B 0.000, C 0.000 }
gfCNCPoint5[19554] = {X 248.7287, Y 8.0298, Z -7.1667, A 0.000, B 0.000, C 0.000 }
gfCNCPoint5[19555] = {X 250.8346, Y 7.9496, Z -7.1667, A 0.000, B 0.000, C 0.000 }
gfCNCPoint5[19556] = {X 266.7627, Y 7.9496, Z -7.1667, A 0.000, B 0.000, C 0.000 }
gfCNCPoint5[19557] = {X 267.7004, Y 8.0622, Z -7.1667, A 0.000, B 0.000, C 0.000 }
gfCNCPoint5[19558] = {X 268.5899, Y 8.3795, Z -7.1667, A 0.000, B 0.000, C 0.000 }
gfCNCPoint5[19559] = {X 269.3872, Y 8.8857, Z -7.1667, A 0.000, B 0.000, C 0.000 }
gfCNCPoint5[19560] = {X 270.0527, Y 9.5558, Z -7.1667, A 0.000, B 0.000, C 0.000 }
gfCNCPoint5[19561] = {X 270.5535, Y 10.3565, Z -7.1667, A 0.000, B 0.000, C 0.000 }
gfCNCPoint5[19562] = {X 270.8647, Y 11.2481, Z -7.1667, A 0.000, B 0.000, C 0.000 }
gfCNCPoint5[19563] = {X 270.9710, Y 12.1865, Z -7.1667, A 0.000, B 0.000, C 0.000 }
gfCNCPoint5[19564] = {X 270.9708, Y 13.0217, Z -7.1667, A 0.000, B 0.000, C 0.000 }
gfCNCPoint5[19565] = {X 270.8625, Y 13.9314, Z -7.1667, A 0.000, B 0.000, C 0.000 }
gfCNCPoint5[19566] = {X 270.5612, Y 14.7966, Z -7.1667, A 0.000, B 0.000, C 0.000 }
gfCNCPoint5[19567] = {X 270.0811, Y 15.5769, Z -7.1667, A 0.000, B 0.000, C 0.000 }
gfCNCPoint5[19568] = {X 269.4447, Y 16.2359, Z -7.1667, A 0.000, B 0.000, C 0.000 }
gfCNCPoint5[19569] = {X 269.4447, Y 28.5937, Z -7.1667, A 0.000, B 0.000, C 0.000 }
gfCNCPoint5[19570] = {X 273.4447, Y 28.5936, Z -7.1667, A 0.000, B 0.000, C 0.000 }
gfCNCPoint5[19571] = {X 269.3647, Y 28.5937, Z -7.1667, A 0.000, B 0.000, C 0.000 }
gfCNCPoint5[19572] = {X 269.3648, Y 40.9897, Z -7.1667, A 0.000, B 0.000, C 0.000 }
gfCNCPoint5[19573] = {X 269.4353, Y 41.0477, Z -7.1667, A 0.000, B 0.000, C 0.000 }
gfCNCPoint5[19574] = {X 270.0436, Y 41.6923, Z -7.1667, A 0.000, B 0.000, C 0.000 }
gfCNCPoint5[19575] = {X 270.5015, Y 42.4511, Z -7.1667, A 0.000, B 0.000, C 0.000 }
gfCNCPoint5[19576] = {X 270.7882, Y 43.2897, Z -7.1667, A 0.000, B 0.000, C 0.000 }
gfCNCPoint5[19577] = {X 270.8909, Y 44.1700, Z -7.1667, A 0.000, B 0.000, C 0.000 }
gfCNCPoint5[19578] = {X 270.8910, Y 45.0000, Z -7.1667, A 0.000, B 0.000, C 0.000 }
gfCNCPoint5[19579] = {X 270.7867, Y 45.9257, Z -7.1667, A 0.000, B 0.000, C 0.000 }
gfCNCPoint5[19580] = {X 270.4791, Y 46.8050, Z -7.1667, A 0.000, B 0.000, C 0.000 }
gfCNCPoint5[19581] = {X 269.9835, Y 47.5937, Z -7.1667, A 0.000, B 0.000, C 0.000 }
gfCNCPoint5[19582] = {X 269.3247, Y 48.2524, Z -7.1667, A 0.000, B 0.000, C 0.000 }
gfCNCPoint5[19583] = {X 268.5360, Y 48.7480, Z -7.1667, A 0.000, B 0.000, C 0.000 }
gfCNCPoint5[19584] = {X 267.6567, Y 49.0557, Z -7.1667, A 0.000, B 0.000, C 0.000 }
gfCNCPoint5[19585] = {X 266.7310, Y 49.1600, Z -7.1667, A 0.000, B 0.000, C 0.000 }
gfCNCPoint5[19586] = {X 260.2876, Y 49.1600, Z -7.1667, A 0.000, B 0.000, C 0.000 }
gfCNCPoint5[19587] = {X 259.3664, Y 49.0567, Z -7.1667, A 0.000, B 0.000, C 0.000 }
gfCNCPoint5[19588] = {X 258.4910, Y 48.7520, Z -7.1667, A 0.000, B 0.000, C 0.000 }
gfCNCPoint5[19589] = {X 257.7047, Y 48.2611, Z -7.1667, A 0.000, B 0.000, C 0.000 }
gfCNCPoint5[19590] = {X 257.0467, Y 47.6082, Z -7.1667, A 0.000, B 0.000, C 0.000 }
gfCNCPoint5[19591] = {X 256.5496, Y 46.8258, Z -7.1667, A 0.000, B 0.000, C 0.000 }
gfCNCPoint5[19592] = {X 256.2381, Y 45.9527, Z -7.1667, A 0.000, B 0.000, C 0.000 }
gfCNCPoint5[19593] = {X 256.1277, Y 45.0324, Z -7.1667, A 0.000, B 0.000, C 0.000 }
gfCNCPoint5[19594] = {X 256.1280, Y 44.1516, Z -7.1667, A 0.000, B 0.000, C 0.000 }
gfCNCPoint5[19595] = {X 256.2385, Y 43.2545, Z -7.1667, A 0.000, B 0.000, C 0.000 }
gfCNCPoint5[19596] = {X 256.5401, Y 42.4026, Z -7.1667, A 0.000, B 0.000, C 0.000 }
gfCNCPoint5[19597] = {X 257.0187, Y 41.6358, Z -7.1667, A 0.000, B 0.000, C 0.000 }
gfCNCPoint5[19598] = {X 257.6515, Y 40.9906, Z -7.1667, A 0.000, B 0.000, C 0.000 }
gfCNCPoint5[19599] = {X 257.6515, Y 34.3138, Z -7.1667, A 0.000, B 0.000, C 0.000 }
gfCNCPoint5[19600] = {X 254.6709, Y 34.3138, Z -7.1667, A 0.000, B 0.000, C 0.000 }
gfCNCPoint5[19601] = {X 250.3103, Y 42.8072, Z -7.1667, A 0.000, B 0.000, C 0.000 }
gfCNCPoint5[19602] = {X 250.4893, Y 43.4802, Z -7.1667, A 0.000, B 0.000, C 0.000 }
gfCNCPoint5[19603] = {X 250.5534, Y 44.1736, Z -7.1667, A 0.000, B 0.000, C 0.000 }
gfCNCPoint5[19604] = {X 250.5536, Y 45.0000, Z -7.1667, A 0.000, B 0.000, C 0.000 }
gfCNCPoint5[19605] = {X 250.4493, Y 45.9257, Z -7.1667, A 0.000, B 0.000, C 0.000 }
gfCNCPoint5[19606] = {X 250.1416, Y 46.8050, Z -7.1667, A 0.000, B 0.000, C 0.000 }
gfCNCPoint5[19607] = {X 249.6460, Y 47.5937, Z -7.1667, A 0.000, B 0.000, C 0.000 }
gfCNCPoint5[19608] = {X 248.9873, Y 48.2524, Z -7.1667, A 0.000, B 0.000, C 0.000 }
gfCNCPoint5[19609] = {X 248.1985, Y 48.7480, Z -7.1667, A 0.000, B 0.000, C 0.000 }
gfCNCPoint5[19610] = {X 247.3192, Y 49.0557, Z -7.1667, A 0.000, B 0.000, C 0.000 }
gfCNCPoint5[19611] = {X 246.3936, Y 49.1600, Z -7.1667, A 0.000, B 0.000, C 0.000 }
gfCNCPoint5[19612] = {X 239.8075, Y 49.1600, Z -7.1667, A 0.000, B 0.000, C 0.000 }
gfCNCPoint5[19613] = {X 238.8818, Y 49.0557, Z -7.1667, A 0.000, B 0.000, C 0.000 }
gfCNCPoint5[19614] = {X 238.0026, Y 48.7480, Z -7.1667, A 0.000, B 0.000, C 0.000 }
gfCNCPoint5[19615] = {X 237.2138, Y 48.2524, Z -7.1667, A 0.000, B 0.000, C 0.000 }
gfCNCPoint5[19616] = {X 236.5551, Y 47.5937, Z -7.1667, A 0.000, B 0.000, C 0.000 }
gfCNCPoint5[19617] = {X 236.0595, Y 46.8050, Z -7.1667, A 0.000, B 0.000, C 0.000 }
gfCNCPoint5[19618] = {X 235.7518, Y 45.9257, Z -7.1667, A 0.000, B 0.000, C 0.000 }
gfCNCPoint5[19619] = {X 235.6475, Y 45.0000, Z -7.1667, A 0.000, B 0.000, C 0.000 }
gfCNCPoint5[19620] = {X 235.6479, Y 44.1516, Z -7.1667, A 0.000, B 0.000, C 0.000 }
gfCNCPoint5[19621] = {X 235.7441, Y 43.3174, Z -7.1667, A 0.000, B 0.000, C 0.000 }
gfCNCPoint5[19622] = {X 236.0059, Y 42.5195, Z -7.1667, A 0.000, B 0.000, C 0.000 }
gfCNCPoint5[19623] = {X 236.4226, Y 41.7905, Z -7.1667, A 0.000, B 0.000, C 0.000 }
gfCNCPoint5[19624] = {X 236.9772, Y 41.1600, Z -7.1667, A 0.000, B 0.000, C 0.000 }
gfCNCPoint5[19625] = {X 237.6471, Y 40.6537, Z -7.1667, A 0.000, B 0.000, C 0.000 }
gfCNCPoint5[19626] = {X 238.4051, Y 40.2923, Z -7.1667, A 0.000, B 0.000, C 0.000 }
gfCNCPoint5[19627] = {X 242.4916, Y 32.2935, Z -7.1667, A 0.000, B 0.000, C 0.000 }
gfCNCPoint5[19628] = {X 241.3075, Y 31.5186, Z -7.1667, A 0.000, B 0.000, C 0.000 }
gfCNCPoint5[19629] = {X 240.2310, Y 30.6001, Z -7.1667, A 0.000, B 0.000, C 0.000 }
gfCNCPoint5[19630] = {X 239.2793, Y 29.5529, Z -7.1667, A 0.000, B 0.000, C 0.000 }
gfCNCPoint5[19631] = {X 238.4677, Y 28.3936, Z -7.1667, A 0.000, B 0.000, C 0.000 }
gfCNCPoint5[19632] = {X 237.8094, Y 27.1410, Z -7.1667, A 0.000, B 0.000, C 0.000 }
gfCNCPoint5[19633] = {X 237.3148, Y 25.8152, Z -7.1667, A 0.000, B 0.000, C 0.000 }
gfCNCPoint5[19634] = {X 236.8989, Y 24.0215, Z -7.1667, A 0.000, B 0.000, C 0.000 }
gfCNCPoint5[19635] = {X 236.6870, Y 22.1924, Z -7.1667, A 0.000, B 0.000, C 0.000 }
gfCNCPoint5[19636] = {X 236.6818, Y 20.3511, Z -7.1667, A 0.000, B 0.000, C 0.000 }
gfCNCPoint5[19637] = {X 236.8833, Y 18.5209, Z -7.1667, A 0.000, B 0.000, C 0.000 }
gfCNCPoint5[19638] = {X 237.2890, Y 16.7248, Z -7.1667, A 0.000, B 0.000, C 0.000 }
gfCNCPoint5[19639] = {X 237.8519, Y 15.1702, Z -7.1667, A 0.000, B 0.000, C 0.000 }
gfCNCPoint5[19640] = {X 238.6284, Y 13.7104, Z -7.1667, A 0.000, B 0.000, C 0.000 }
gfCNCPoint5[19641] = {X 239.6032, Y 12.3749, Z -7.1667, A 0.000, B 0.000, C 0.000 }
gfCNCPoint5[19642] = {X 240.7566, Y 11.1902, Z -7.1667, A 0.000, B 0.000, C 0.000 }
gfCNCPoint5[19643] = {X 242.0656, Y 10.1800, Z -7.1667, A 0.000, B 0.000, C 0.000 }
gfCNCPoint5[19644] = {X 243.5040, Y 9.3647, Z -7.1667, A 0.000, B 0.000, C 0.000 }
gfCNCPoint5[19645] = {X 245.0430, Y 8.7604, Z -7.1667, A 0.000, B 0.000, C 0.000 }
gfCNCPoint5[19646] = {X 246.6520, Y 8.3793, Z -7.1667, A 0.000, B 0.000, C 0.000 }
gfCNCPoint5[19647] = {X 248.7352, Y 8.1096, Z -7.1667, A 0.000, B 0.000, C 0.000 }
gfCNCPoint5[19648] = {X 250.8343, Y 8.0296, Z -7.1667, A 0.000, B 0.000, C 0.000 }
gfCNCPoint5[19649] = {X 266.7621, Y 8.0296, Z -7.1667, A 0.000, B 0.000, C 0.000 }
gfCNCPoint5[19650] = {X 267.6820, Y 8.1401, Z -7.1667, A 0.000, B 0.000, C 0.000 }
gfCNCPoint5[19651] = {X 268.5548, Y 8.4514, Z -7.1667, A 0.000, B 0.000, C 0.000 }
gfCNCPoint5[19652] = {X 269.3370, Y 8.9481, Z -7.1667, A 0.000, B 0.000, C 0.000 }
gfCNCPoint5[19653] = {X 269.9900, Y 9.6055, Z -7.1667, A 0.000, B 0.000, C 0.000 }
gfCNCPoint5[19654] = {X 270.4814, Y 10.3911, Z -7.1667, A 0.000, B 0.000, C 0.000 }
gfCNCPoint5[19655] = {X 270.7868, Y 11.2659, Z -7.1667, A 0.000, B 0.000, C 0.000 }
gfCNCPoint5[19656] = {X 270.8910, Y 12.1866, Z -7.1667, A 0.000, B 0.000, C 0.000 }
gfCNCPoint5[19657] = {X 270.8908, Y 13.0208, Z -7.1667, A 0.000, B 0.000, C 0.000 }
gfCNCPoint5[19658] = {X 270.7824, Y 13.9225, Z -7.1667, A 0.000, B 0.000, C 0.000 }
gfCNCPoint5[19659] = {X 270.4809, Y 14.7792, Z -7.1667, A 0.000, B 0.000, C 0.000 }
gfCNCPoint5[19660] = {X 270.0007, Y 15.5500, Z -7.1667, A 0.000, B 0.000, C 0.000 }
gfCNCPoint5[19661] = {X 269.3647, Y 16.1982, Z -7.1667, A 0.000, B 0.000, C 0.000 }
gfCNCPoint5[19662] = {X 269.3647, Y 28.5937, Z -7.1667, A 0.000, B 0.000, C 0.000 }
gfCNCPoint5[19663] = {X 273.3647, Y 28.5936, Z -7.1667, A 0.000, B 0.000, C 0.000 }
gfCNCPoint5[19664] = {X 269.2847, Y 28.5937, Z -7.1667, A 0.000, B 0.000, C 0.000 }
gfCNCPoint5[19665] = {X 269.2848, Y 41.0276, Z -7.1667, A 0.000, B 0.000, C 0.000 }
gfCNCPoint5[19666] = {X 269.3839, Y 41.1090, Z -7.1667, A 0.000, B 0.000, C 0.000 }
gfCNCPoint5[19667] = {X 269.9802, Y 41.7412, Z -7.1667, A 0.000, B 0.000, C 0.000 }
gfCNCPoint5[19668] = {X 270.4291, Y 42.4853, Z -7.1667, A 0.000, B 0.000, C 0.000 }
gfCNCPoint5[19669] = {X 270.7103, Y 43.3076, Z -7.1667, A 0.000, B 0.000, C 0.000 }
gfCNCPoint5[19670] = {X 270.8109, Y 44.1708, Z -7.1667, A 0.000, B 0.000, C 0.000 }
gfCNCPoint5[19671] = {X 270.8110, Y 45.0000, Z -7.1667, A 0.000, B 0.000, C 0.000 }
gfCNCPoint5[19672] = {X 270.7087, Y 45.9079, Z -7.1667, A 0.000, B 0.000, C 0.000 }
gfCNCPoint5[19673] = {X 270.4070, Y 46.7702, Z -7.1667, A 0.000, B 0.000, C 0.000 }
gfCNCPoint5[19674] = {X 269.9209, Y 47.5438, Z -7.1667, A 0.000, B 0.000, C 0.000 }
gfCNCPoint5[19675] = {X 269.2749, Y 48.1899, Z -7.1667, A 0.000, B 0.000, C 0.000 }
gfCNCPoint5[19676] = {X 268.5013, Y 48.6760, Z -7.1667, A 0.000, B 0.000, C 0.000 }
gfCNCPoint5[19677] = {X 267.6389, Y 48.9777, Z -7.1667, A 0.000, B 0.000, C 0.000 }
gfCNCPoint5[19678] = {X 266.7310, Y 49.0800, Z -7.1667, A 0.000, B 0.000, C 0.000 }
gfCNCPoint5[19679] = {X 260.2876, Y 49.0800, Z -7.1667, A 0.000, B 0.000, C 0.000 }
gfCNCPoint5[19680] = {X 259.3841, Y 48.9787, Z -7.1667, A 0.000, B 0.000, C 0.000 }
gfCNCPoint5[19681] = {X 258.5255, Y 48.6799, Z -7.1667, A 0.000, B 0.000, C 0.000 }
gfCNCPoint5[19682] = {X 257.7544, Y 48.1983, Z -7.1667, A 0.000, B 0.000, C 0.000 }
gfCNCPoint5[19683] = {X 257.1090, Y 47.5580, Z -7.1667, A 0.000, B 0.000, C 0.000 }
gfCNCPoint5[19684] = {X 256.6215, Y 46.7907, Z -7.1667, A 0.000, B 0.000, C 0.000 }
gfCNCPoint5[19685] = {X 256.3160, Y 45.9344, Z -7.1667, A 0.000, B 0.000, C 0.000 }
gfCNCPoint5[19686] = {X 256.2077, Y 45.0318, Z -7.1667, A 0.000, B 0.000, C 0.000 }
gfCNCPoint5[19687] = {X 256.2080, Y 44.1527, Z -7.1667, A 0.000, B 0.000, C 0.000 }
gfCNCPoint5[19688] = {X 256.3185, Y 43.2637, Z -7.1667, A 0.000, B 0.000, C 0.000 }
gfCNCPoint5[19689] = {X 256.6204, Y 42.4203, Z -7.1667, A 0.000, B 0.000, C 0.000 }
gfCNCPoint5[19690] = {X 257.0991, Y 41.6631, Z -7.1667, A 0.000, B 0.000, C 0.000 }
gfCNCPoint5[19691] = {X 257.7315, Y 41.0287, Z -7.1667, A 0.000, B 0.000, C 0.000 }
gfCNCPoint5[19692] = {X 257.7315, Y 34.2338, Z -7.1667, A 0.000, B 0.000, C 0.000 }
gfCNCPoint5[19693] = {X 254.6221, Y 34.2338, Z -7.1667, A 0.000, B 0.000, C 0.000 }
gfCNCPoint5[19694] = {X 250.2232, Y 42.8017, Z -7.1667, A 0.000, B 0.000, C 0.000 }
gfCNCPoint5[19695] = {X 250.4074, Y 43.4772, Z -7.1667, A 0.000, B 0.000, C 0.000 }
gfCNCPoint5[19696] = {X 250.4734, Y 44.1743, Z -7.1667, A 0.000, B 0.000, C 0.000 }
gfCNCPoint5[19697] = {X 250.4736, Y 45.0000, Z -7.1667, A 0.000, B 0.000, C 0.000 }
gfCNCPoint5[19698] = {X 250.3713, Y 45.9079, Z -7.1667, A 0.000, B 0.000, C 0.000 }
gfCNCPoint5[19699] = {X 250.0695, Y 46.7702, Z -7.1667, A 0.000, B 0.000, C 0.000 }
gfCNCPoint5[19700] = {X 249.5834, Y 47.5438, Z -7.1667, A 0.000, B 0.000, C 0.000 }
gfCNCPoint5[19701] = {X 248.9374, Y 48.1899, Z -7.1667, A 0.000, B 0.000, C 0.000 }
gfCNCPoint5[19702] = {X 248.1638, Y 48.6760, Z -7.1667, A 0.000, B 0.000, C 0.000 }
gfCNCPoint5[19703] = {X 247.3014, Y 48.9777, Z -7.1667, A 0.000, B 0.000, C 0.000 }
gfCNCPoint5[19704] = {X 246.3936, Y 49.0800, Z -7.1667, A 0.000, B 0.000, C 0.000 }
gfCNCPoint5[19705] = {X 239.8075, Y 49.0800, Z -7.1667, A 0.000, B 0.000, C 0.000 }
gfCNCPoint5[19706] = {X 238.8996, Y 48.9777, Z -7.1667, A 0.000, B 0.000, C 0.000 }
gfCNCPoint5[19707] = {X 238.0373, Y 48.6760, Z -7.1667, A 0.000, B 0.000, C 0.000 }
gfCNCPoint5[19708] = {X 237.2637, Y 48.1899, Z -7.1667, A 0.000, B 0.000, C 0.000 }
gfCNCPoint5[19709] = {X 236.6176, Y 47.5438, Z -7.1667, A 0.000, B 0.000, C 0.000 }
gfCNCPoint5[19710] = {X 236.1315, Y 46.7702, Z -7.1667, A 0.000, B 0.000, C 0.000 }
gfCNCPoint5[19711] = {X 235.8298, Y 45.9079, Z -7.1667, A 0.000, B 0.000, C 0.000 }
gfCNCPoint5[19712] = {X 235.7275, Y 45.0000, Z -7.1667, A 0.000, B 0.000, C 0.000 }
gfCNCPoint5[19713] = {X 235.7279, Y 44.1527, Z -7.1667, A 0.000, B 0.000, C 0.000 }
gfCNCPoint5[19714] = {X 235.8234, Y 43.3294, Z -7.1667, A 0.000, B 0.000, C 0.000 }
gfCNCPoint5[19715] = {X 236.0833, Y 42.5424, Z -7.1667, A 0.000, B 0.000, C 0.000 }
gfCNCPoint5[19716] = {X 236.4969, Y 41.8242, Z -7.1667, A 0.000, B 0.000, C 0.000 }
gfCNCPoint5[19717] = {X 237.0471, Y 41.2044, Z -7.1667, A 0.000, B 0.000, C 0.000 }
gfCNCPoint5[19718] = {X 237.7112, Y 40.7085, Z -7.1667, A 0.000, B 0.000, C 0.000 }
gfCNCPoint5[19719] = {X 238.4618, Y 40.3571, Z -7.1667, A 0.000, B 0.000, C 0.000 }
gfCNCPoint5[19720] = {X 242.5978, Y 32.2614, Z -7.1667, A 0.000, B 0.000, C 0.000 }
gfCNCPoint5[19721] = {X 241.4066, Y 31.4927, Z -7.1667, A 0.000, B 0.000, C 0.000 }
gfCNCPoint5[19722] = {X 240.3234, Y 30.5781, Z -7.1667, A 0.000, B 0.000, C 0.000 }
gfCNCPoint5[19723] = {X 239.3657, Y 29.5328, Z -7.1667, A 0.000, B 0.000, C 0.000 }
gfCNCPoint5[19724] = {X 238.5493, Y 28.3738, Z -7.1667, A 0.000, B 0.000, C 0.000 }
gfCNCPoint5[19725] = {X 237.8876, Y 27.1200, Z -7.1667, A 0.000, B 0.000, C 0.000 }
gfCNCPoint5[19726] = {X 237.3913, Y 25.7920, Z -7.1667, A 0.000, B 0.000, C 0.000 }
gfCNCPoint5[19727] = {X 236.9776, Y 24.0072, Z -7.1667, A 0.000, B 0.000, C 0.000 }
gfCNCPoint5[19728] = {X 236.7668, Y 22.1872, Z -7.1667, A 0.000, B 0.000, C 0.000 }
gfCNCPoint5[19729] = {X 236.7617, Y 20.3551, Z -7.1667, A 0.000, B 0.000, C 0.000 }
gfCNCPoint5[19730] = {X 236.9622, Y 18.5339, Z -7.1667, A 0.000, B 0.000, C 0.000 }
gfCNCPoint5[19731] = {X 237.3660, Y 16.7468, Z -7.1667, A 0.000, B 0.000, C 0.000 }
gfCNCPoint5[19732] = {X 237.9250, Y 15.2027, Z -7.1667, A 0.000, B 0.000, C 0.000 }
gfCNCPoint5[19733] = {X 238.6963, Y 13.7529, Z -7.1667, A 0.000, B 0.000, C 0.000 }
gfCNCPoint5[19734] = {X 239.6644, Y 12.4264, Z -7.1667, A 0.000, B 0.000, C 0.000 }
gfCNCPoint5[19735] = {X 240.8099, Y 11.2498, Z -7.1667, A 0.000, B 0.000, C 0.000 }
gfCNCPoint5[19736] = {X 242.1101, Y 10.2465, Z -7.1667, A 0.000, B 0.000, C 0.000 }
gfCNCPoint5[19737] = {X 243.5387, Y 9.4367, Z -7.1667, A 0.000, B 0.000, C 0.000 }
gfCNCPoint5[19738] = {X 245.0673, Y 8.8366, Z -7.1667, A 0.000, B 0.000, C 0.000 }
gfCNCPoint5[19739] = {X 246.6653, Y 8.4582, Z -7.1667, A 0.000, B 0.000, C 0.000 }
gfCNCPoint5[19740] = {X 248.7417, Y 8.1893, Z -7.1667, A 0.000, B 0.000, C 0.000 }
gfCNCPoint5[19741] = {X 250.8340, Y 8.1096, Z -7.1667, A 0.000, B 0.000, C 0.000 }
gfCNCPoint5[19742] = {X 266.7614, Y 8.1096, Z -7.1667, A 0.000, B 0.000, C 0.000 }
gfCNCPoint5[19743] = {X 267.6637, Y 8.2180, Z -7.1667, A 0.000, B 0.000, C 0.000 }
gfCNCPoint5[19744] = {X 268.5197, Y 8.5233, Z -7.1667, A 0.000, B 0.000, C 0.000 }
gfCNCPoint5[19745] = {X 269.2869, Y 9.0104, Z -7.1667, A 0.000, B 0.000, C 0.000 }
gfCNCPoint5[19746] = {X 269.9273, Y 9.6552, Z -7.1667, A 0.000, B 0.000, C 0.000 }
gfCNCPoint5[19747] = {X 270.4092, Y 10.4257, Z -7.1667, A 0.000, B 0.000, C 0.000 }
gfCNCPoint5[19748] = {X 270.7088, Y 11.2837, Z -7.1667, A 0.000, B 0.000, C 0.000 }
gfCNCPoint5[19749] = {X 270.8110, Y 12.1867, Z -7.1667, A 0.000, B 0.000, C 0.000 }
gfCNCPoint5[19750] = {X 270.8108, Y 13.0200, Z -7.1667, A 0.000, B 0.000, C 0.000 }
gfCNCPoint5[19751] = {X 270.7023, Y 13.9135, Z -7.1667, A 0.000, B 0.000, C 0.000 }
gfCNCPoint5[19752] = {X 270.4006, Y 14.7615, Z -7.1667, A 0.000, B 0.000, C 0.000 }
gfCNCPoint5[19753] = {X 269.9202, Y 15.5227, Z -7.1667, A 0.000, B 0.000, C 0.000 }
gfCNCPoint5[19754] = {X 269.2847, Y 16.1601, Z -7.1667, A 0.000, B 0.000, C 0.000 }
gfCNCPoint5[19755] = {X 269.2847, Y 28.5937, Z -7.1667, A 0.000, B 0.000, C 0.000 }
gfCNCPoint5[19756] = {X 273.2847, Y 28.5936, Z -7.1667, A 0.000, B 0.000, C 0.000 }
gfCNCPoint5[19757] = {X 269.2047, Y 28.5937, Z -7.1667, A 0.000, B 0.000, C 0.000 }
gfCNCPoint5[19758] = {X 269.2048, Y 41.0654, Z -7.1667, A 0.000, B 0.000, C 0.000 }
gfCNCPoint5[19759] = {X 269.3435, Y 41.1798, Z -7.1667, A 0.000, B 0.000, C 0.000 }
gfCNCPoint5[19760] = {X 269.9291, Y 41.8062, Z -7.1667, A 0.000, B 0.000, C 0.000 }
gfCNCPoint5[19761] = {X 270.3677, Y 42.5430, Z -7.1667, A 0.000, B 0.000, C 0.000 }
gfCNCPoint5[19762] = {X 270.6391, Y 43.3563, Z -7.1667, A 0.000, B 0.000, C 0.000 }
gfCNCPoint5[19763] = {X 270.7310, Y 44.2089, Z -7.1667, A 0.000, B 0.000, C 0.000 }
gfCNCPoint5[19764] = {X 270.7310, Y 45.0000, Z -7.1667, A 0.000, B 0.000, C 0.000 }
gfCNCPoint5[19765] = {X 270.6307, Y 45.8901, Z -7.1667, A 0.000, B 0.000, C 0.000 }
gfCNCPoint5[19766] = {X 270.3349, Y 46.7355, Z -7.1667, A 0.000, B 0.000, C 0.000 }
gfCNCPoint5[19767] = {X 269.8584, Y 47.4940, Z -7.1667, A 0.000, B 0.000, C 0.000 }
gfCNCPoint5[19768] = {X 269.2250, Y 48.1273, Z -7.1667, A 0.000, B 0.000, C 0.000 }
gfCNCPoint5[19769] = {X 268.4666, Y 48.6039, Z -7.1667, A 0.000, B 0.000, C 0.000 }
gfCNCPoint5[19770] = {X 267.6211, Y 48.8997, Z -7.1667, A 0.000, B 0.000, C 0.000 }
gfCNCPoint5[19771] = {X 266.7310, Y 49.0000, Z -7.1667, A 0.000, B 0.000, C 0.000 }
gfCNCPoint5[19772] = {X 260.2876, Y 49.0000, Z -7.1667, A 0.000, B 0.000, C 0.000 }
gfCNCPoint5[19773] = {X 259.3975, Y 48.8997, Z -7.1667, A 0.000, B 0.000, C 0.000 }
gfCNCPoint5[19774] = {X 258.5520, Y 48.6039, Z -7.1667, A 0.000, B 0.000, C 0.000 }
gfCNCPoint5[19775] = {X 257.7936, Y 48.1273, Z -7.1667, A 0.000, B 0.000, C 0.000 }
gfCNCPoint5[19776] = {X 257.1602, Y 47.4939, Z -7.1667, A 0.000, B 0.000, C 0.000 }
gfCNCPoint5[19777] = {X 256.6837, Y 46.7355, Z -7.1667, A 0.000, B 0.000, C 0.000 }
gfCNCPoint5[19778] = {X 256.3878, Y 45.8901, Z -7.1667, A 0.000, B 0.000, C 0.000 }
gfCNCPoint5[19779] = {X 256.2876, Y 45.0000, Z -7.1667, A 0.000, B 0.000, C 0.000 }
gfCNCPoint5[19780] = {X 256.2879, Y 44.1538, Z -7.1667, A 0.000, B 0.000, C 0.000 }
gfCNCPoint5[19781] = {X 256.3986, Y 43.2730, Z -7.1667, A 0.000, B 0.000, C 0.000 }
gfCNCPoint5[19782] = {X 256.7008, Y 42.4382, Z -7.1667, A 0.000, B 0.000, C 0.000 }
gfCNCPoint5[19783] = {X 257.1796, Y 41.6907, Z -7.1667, A 0.000, B 0.000, C 0.000 }
gfCNCPoint5[19784] = {X 257.8115, Y 41.0672, Z -7.1667, A 0.000, B 0.000, C 0.000 }
gfCNCPoint5[19785] = {X 257.8115, Y 34.1538, Z -7.1667, A 0.000, B 0.000, C 0.000 }
gfCNCPoint5[19786] = {X 254.8175, Y 34.1538, Z -7.1667, A 0.000, B 0.000, C 0.000 }
gfCNCPoint5[19787] = {X 254.5736, Y 34.1531, Z -7.1667, A 0.000, B 0.000, C 0.000 }
gfCNCPoint5[19788] = {X 250.1359, Y 42.7965, Z -7.1667, A 0.000, B 0.000, C 0.000 }
gfCNCPoint5[19789] = {X 250.3286, Y 43.4910, Z -7.1667, A 0.000, B 0.000, C 0.000 }
gfCNCPoint5[19790] = {X 250.3936, Y 44.2089, Z -7.1667, A 0.000, B 0.000, C 0.000 }
gfCNCPoint5[19791] = {X 250.3936, Y 45.0000, Z -7.1667, A 0.000, B 0.000, C 0.000 }
gfCNCPoint5[19792] = {X 250.2933, Y 45.8901, Z -7.1667, A 0.000, B 0.000, C 0.000 }
gfCNCPoint5[19793] = {X 249.9974, Y 46.7355, Z -7.1667, A 0.000, B 0.000, C 0.000 }
gfCNCPoint5[19794] = {X 249.5209, Y 47.4940, Z -7.1667, A 0.000, B 0.000, C 0.000 }
gfCNCPoint5[19795] = {X 248.8875, Y 48.1273, Z -7.1667, A 0.000, B 0.000, C 0.000 }
gfCNCPoint5[19796] = {X 248.1291, Y 48.6039, Z -7.1667, A 0.000, B 0.000, C 0.000 }
gfCNCPoint5[19797] = {X 247.2836, Y 48.8997, Z -7.1667, A 0.000, B 0.000, C 0.000 }
gfCNCPoint5[19798] = {X 246.3936, Y 49.0000, Z -7.1667, A 0.000, B 0.000, C 0.000 }
gfCNCPoint5[19799] = {X 239.8075, Y 49.0000, Z -7.1667, A 0.000, B 0.000, C 0.000 }
gfCNCPoint5[19800] = {X 238.9174, Y 48.8997, Z -7.1667, A 0.000, B 0.000, C 0.000 }
gfCNCPoint5[19801] = {X 238.0720, Y 48.6039, Z -7.1667, A 0.000, B 0.000, C 0.000 }
gfCNCPoint5[19802] = {X 237.3135, Y 48.1273, Z -7.1667, A 0.000, B 0.000, C 0.000 }
gfCNCPoint5[19803] = {X 236.6802, Y 47.4940, Z -7.1667, A 0.000, B 0.000, C 0.000 }
gfCNCPoint5[19804] = {X 236.2036, Y 46.7355, Z -7.1667, A 0.000, B 0.000, C 0.000 }
gfCNCPoint5[19805] = {X 235.9078, Y 45.8901, Z -7.1667, A 0.000, B 0.000, C 0.000 }
gfCNCPoint5[19806] = {X 235.8075, Y 45.0000, Z -7.1667, A 0.000, B 0.000, C 0.000 }
gfCNCPoint5[19807] = {X 235.8079, Y 44.1538, Z -7.1667, A 0.000, B 0.000, C 0.000 }
gfCNCPoint5[19808] = {X 235.9027, Y 43.3414, Z -7.1667, A 0.000, B 0.000, C 0.000 }
gfCNCPoint5[19809] = {X 236.1607, Y 42.5654, Z -7.1667, A 0.000, B 0.000, C 0.000 }
gfCNCPoint5[19810] = {X 236.5712, Y 41.8580, Z -7.1667, A 0.000, B 0.000, C 0.000 }
gfCNCPoint5[19811] = {X 237.1169, Y 41.2489, Z -7.1667, A 0.000, B 0.000, C 0.000 }
gfCNCPoint5[19812] = {X 237.7752, Y 40.7635, Z -7.1667, A 0.000, B 0.000, C 0.000 }
gfCNCPoint5[19813] = {X 238.5184, Y 40.4222, Z -7.1667, A 0.000, B 0.000, C 0.000 }
gfCNCPoint5[19814] = {X 242.7042, Y 32.2289, Z -7.1667, A 0.000, B 0.000, C 0.000 }
gfCNCPoint5[19815] = {X 241.5060, Y 31.4664, Z -7.1667, A 0.000, B 0.000, C 0.000 }
gfCNCPoint5[19816] = {X 240.4159, Y 30.5559, Z -7.1667, A 0.000, B 0.000, C 0.000 }
gfCNCPoint5[19817] = {X 239.4523, Y 29.5126, Z -7.1667, A 0.000, B 0.000, C 0.000 }
gfCNCPoint5[19818] = {X 238.6310, Y 28.3539, Z -7.1667, A 0.000, B 0.000, C 0.000 }
gfCNCPoint5[19819] = {X 237.9659, Y 27.0990, Z -7.1667, A 0.000, B 0.000, C 0.000 }
gfCNCPoint5[19820] = {X 237.4679, Y 25.7689, Z -7.1667, A 0.000, B 0.000, C 0.000 }
gfCNCPoint5[19821] = {X 237.0563, Y 23.9929, Z -7.1667, A 0.000, B 0.000, C 0.000 }
gfCNCPoint5[19822] = {X 236.8466, Y 22.1820, Z -7.1667, A 0.000, B 0.000, C 0.000 }
gfCNCPoint5[19823] = {X 236.8416, Y 20.3590, Z -7.1667, A 0.000, B 0.000, C 0.000 }
gfCNCPoint5[19824] = {X 237.0412, Y 18.5469, Z -7.1667, A 0.000, B 0.000, C 0.000 }
gfCNCPoint5[19825] = {X 237.4429, Y 16.7687, Z -7.1667, A 0.000, B 0.000, C 0.000 }
gfCNCPoint5[19826] = {X 237.9981, Y 15.2352, Z -7.1667, A 0.000, B 0.000, C 0.000 }
gfCNCPoint5[19827] = {X 238.7641, Y 13.7953, Z -7.1667, A 0.000, B 0.000, C 0.000 }
gfCNCPoint5[19828] = {X 239.7256, Y 12.4779, Z -7.1667, A 0.000, B 0.000, C 0.000 }
gfCNCPoint5[19829] = {X 240.8633, Y 11.3093, Z -7.1667, A 0.000, B 0.000, C 0.000 }
gfCNCPoint5[19830] = {X 242.1546, Y 10.3130, Z -7.1667, A 0.000, B 0.000, C 0.000 }
gfCNCPoint5[19831] = {X 243.5735, Y 9.5088, Z -7.1667, A 0.000, B 0.000, C 0.000 }
gfCNCPoint5[19832] = {X 245.0917, Y 8.9129, Z -7.1667, A 0.000, B 0.000, C 0.000 }
gfCNCPoint5[19833] = {X 246.6787, Y 8.5371, Z -7.1667, A 0.000, B 0.000, C 0.000 }
gfCNCPoint5[19834] = {X 248.7483, Y 8.2690, Z -7.1667, A 0.000, B 0.000, C 0.000 }
gfCNCPoint5[19835] = {X 250.8336, Y 8.1896, Z -7.1667, A 0.000, B 0.000, C 0.000 }
gfCNCPoint5[19836] = {X 266.7608, Y 8.1896, Z -7.1667, A 0.000, B 0.000, C 0.000 }
gfCNCPoint5[19837] = {X 267.6454, Y 8.2958, Z -7.1667, A 0.000, B 0.000, C 0.000 }
gfCNCPoint5[19838] = {X 268.4846, Y 8.5952, Z -7.1667, A 0.000, B 0.000, C 0.000 }
gfCNCPoint5[19839] = {X 269.2368, Y 9.0728, Z -7.1667, A 0.000, B 0.000, C 0.000 }
gfCNCPoint5[19840] = {X 269.8646, Y 9.7049, Z -7.1667, A 0.000, B 0.000, C 0.000 }
gfCNCPoint5[19841] = {X 270.3371, Y 10.4603, Z -7.1667, A 0.000, B 0.000, C 0.000 }
gfCNCPoint5[19842] = {X 270.6308, Y 11.3015, Z -7.1667, A 0.000, B 0.000, C 0.000 }
gfCNCPoint5[19843] = {X 270.7310, Y 12.1868, Z -7.1667, A 0.000, B 0.000, C 0.000 }
gfCNCPoint5[19844] = {X 270.7308, Y 13.0192, Z -7.1667, A 0.000, B 0.000, C 0.000 }
gfCNCPoint5[19845] = {X 270.6223, Y 13.9045, Z -7.1667, A 0.000, B 0.000, C 0.000 }
gfCNCPoint5[19846] = {X 270.3202, Y 14.7437, Z -7.1667, A 0.000, B 0.000, C 0.000 }
gfCNCPoint5[19847] = {X 269.8397, Y 15.4952, Z -7.1667, A 0.000, B 0.000, C 0.000 }
gfCNCPoint5[19848] = {X 269.2047, Y 16.1215, Z -7.1667, A 0.000, B 0.000, C 0.000 }
gfCNCPoint5[19849] = {X 269.2047, Y 28.5937, Z -7.1667, A 0.000, B 0.000, C 0.000 }
gfCNCPoint5[19850] = {X 273.2847, Y 28.5936, Z -7.1667, A 0.000, B 0.000, C 0.000 }
gfCNCPoint5[19851] = {X 273.2847, Y 28.5936, Z -4.1667, A 0.000, B 0.000, C 0.000 }
gfCNCPoint5[19852] = {X 273.2847, Y 28.5936, Z 11.0000, A 0.000, B 0.000, C 0.000 }
gfCNCPoint5[19853] = {X 277.7444, Y 28.5919, Z 11.0000, A 0.000, B 0.000, C 0.000 }
gfCNCPoint5[19854] = {X 277.7444, Y 28.5919, Z -4.1667, A 0.000, B 0.000, C 0.000 }
gfCNCPoint5[19855] = {X 277.7444, Y 28.5919, Z -7.1667, A 0.000, B 0.000, C 0.000 }
gfCNCPoint5[19856] = {X 281.8244, Y 28.5919, Z -7.1667, A 0.000, B 0.000, C 0.000 }
gfCNCPoint5[19857] = {X 281.8243, Y 16.2734, Z -7.1667, A 0.000, B 0.000, C 0.000 }
gfCNCPoint5[19858] = {X 281.1862, Y 15.6023, Z -7.1667, A 0.000, B 0.000, C 0.000 }
gfCNCPoint5[19859] = {X 280.7057, Y 14.8107, Z -7.1667, A 0.000, B 0.000, C 0.000 }
gfCNCPoint5[19860] = {X 280.4050, Y 13.9349, Z -7.1667, A 0.000, B 0.000, C 0.000 }
gfCNCPoint5[19861] = {X 280.2978, Y 13.0151, Z -7.1667, A 0.000, B 0.000, C 0.000 }
gfCNCPoint5[19862] = {X 280.2977, Y 12.1868, Z -7.1667, A 0.000, B 0.000, C 0.000 }
gfCNCPoint5[19863] = {X 280.4060, Y 11.2255, Z -7.1667, A 0.000, B 0.000, C 0.000 }
gfCNCPoint5[19864] = {X 280.7255, Y 10.3124, Z -7.1667, A 0.000, B 0.000, C 0.000 }
gfCNCPoint5[19865] = {X 281.2402, Y 9.4933, Z -7.1667, A 0.000, B 0.000, C 0.000 }
gfCNCPoint5[19866] = {X 281.9242, Y 8.8093, Z -7.1667, A 0.000, B 0.000, C 0.000 }
gfCNCPoint5[19867] = {X 282.7433, Y 8.2946, Z -7.1667, A 0.000, B 0.000, C 0.000 }
gfCNCPoint5[19868] = {X 283.6564, Y 7.9751, Z -7.1667, A 0.000, B 0.000, C 0.000 }
gfCNCPoint5[19869] = {X 284.6177, Y 7.8668, Z -7.1667, A 0.000, B 0.000, C 0.000 }
gfCNCPoint5[19870] = {X 291.0611, Y 7.8668, Z -7.1667, A 0.000, B 0.000, C 0.000 }
gfCNCPoint5[19871] = {X 292.0224, Y 7.9751, Z -7.1667, A 0.000, B 0.000, C 0.000 }
gfCNCPoint5[19872] = {X 292.9355, Y 8.2946, Z -7.1667, A 0.000, B 0.000, C 0.000 }
gfCNCPoint5[19873] = {X 293.7546, Y 8.8093, Z -7.1667, A 0.000, B 0.000, C 0.000 }
gfCNCPoint5[19874] = {X 294.4386, Y 9.4933, Z -7.1667, A 0.000, B 0.000, C 0.000 }
gfCNCPoint5[19875] = {X 294.9533, Y 10.3124, Z -7.1667, A 0.000, B 0.000, C 0.000 }
gfCNCPoint5[19876] = {X 295.2728, Y 11.2255, Z -7.1667, A 0.000, B 0.000, C 0.000 }
gfCNCPoint5[19877] = {X 295.3811, Y 12.1868, Z -7.1667, A 0.000, B 0.000, C 0.000 }
gfCNCPoint5[19878] = {X 295.3811, Y 12.9782, Z -7.1667, A 0.000, B 0.000, C 0.000 }
gfCNCPoint5[19879] = {X 295.2798, Y 13.9078, Z -7.1667, A 0.000, B 0.000, C 0.000 }
gfCNCPoint5[19880] = {X 294.9808, Y 14.7938, Z -7.1667, A 0.000, B 0.000, C 0.000 }
gfCNCPoint5[19881] = {X 294.4982, Y 15.5947, Z -7.1667, A 0.000, B 0.000, C 0.000 }
gfCNCPoint5[19882] = {X 293.8545, Y 16.2730, Z -7.1667, A 0.000, B 0.000, C 0.000 }
gfCNCPoint5[19883] = {X 293.8554, Y 22.1965, Z -7.1667, A 0.000, B 0.000, C 0.000 }
gfCNCPoint5[19884] = {X 302.7584, Y 22.1965, Z -7.1667, A 0.000, B 0.000, C 0.000 }
gfCNCPoint5[19885] = {X 302.7635, Y 16.2773, Z -7.1667, A 0.000, B 0.000, C 0.000 }
gfCNCPoint5[19886] = {X 302.1237, Y 15.6062, Z -7.1667, A 0.000, B 0.000, C 0.000 }
gfCNCPoint5[19887] = {X 301.6419, Y 14.8141, Z -7.1667, A 0.000, B 0.000, C 0.000 }
gfCNCPoint5[19888] = {X 301.3401, Y 13.9374, Z -7.1667, A 0.000, B 0.000, C 0.000 }
gfCNCPoint5[19889] = {X 301.2324, Y 13.0165, Z -7.1667, A 0.000, B 0.000, C 0.000 }
gfCNCPoint5[19890] = {X 301.2323, Y 12.1868, Z -7.1667, A 0.000, B 0.000, C 0.000 }
gfCNCPoint5[19891] = {X 301.3406, Y 11.2255, Z -7.1667, A 0.000, B 0.000, C 0.000 }
gfCNCPoint5[19892] = {X 301.6601, Y 10.3124, Z -7.1667, A 0.000, B 0.000, C 0.000 }
gfCNCPoint5[19893] = {X 302.1747, Y 9.4933, Z -7.1667, A 0.000, B 0.000, C 0.000 }
gfCNCPoint5[19894] = {X 302.8588, Y 8.8093, Z -7.1667, A 0.000, B 0.000, C 0.000 }
gfCNCPoint5[19895] = {X 303.6779, Y 8.2946, Z -7.1667, A 0.000, B 0.000, C 0.000 }
gfCNCPoint5[19896] = {X 304.5910, Y 7.9751, Z -7.1667, A 0.000, B 0.000, C 0.000 }
gfCNCPoint5[19897] = {X 305.5523, Y 7.8668, Z -7.1667, A 0.000, B 0.000, C 0.000 }
gfCNCPoint5[19898] = {X 311.9957, Y 7.8668, Z -7.1667, A 0.000, B 0.000, C 0.000 }
gfCNCPoint5[19899] = {X 312.9570, Y 7.9751, Z -7.1667, A 0.000, B 0.000, C 0.000 }
gfCNCPoint5[19900] = {X 313.8701, Y 8.2946, Z -7.1667, A 0.000, B 0.000, C 0.000 }
gfCNCPoint5[19901] = {X 314.6892, Y 8.8093, Z -7.1667, A 0.000, B 0.000, C 0.000 }
gfCNCPoint5[19902] = {X 315.3732, Y 9.4933, Z -7.1667, A 0.000, B 0.000, C 0.000 }
gfCNCPoint5[19903] = {X 315.8879, Y 10.3124, Z -7.1667, A 0.000, B 0.000, C 0.000 }
gfCNCPoint5[19904] = {X 316.2074, Y 11.2255, Z -7.1667, A 0.000, B 0.000, C 0.000 }
gfCNCPoint5[19905] = {X 316.3157, Y 12.1868, Z -7.1667, A 0.000, B 0.000, C 0.000 }
gfCNCPoint5[19906] = {X 316.3157, Y 12.9782, Z -7.1667, A 0.000, B 0.000, C 0.000 }
gfCNCPoint5[19907] = {X 316.2145, Y 13.9077, Z -7.1667, A 0.000, B 0.000, C 0.000 }
gfCNCPoint5[19908] = {X 315.9156, Y 14.7937, Z -7.1667, A 0.000, B 0.000, C 0.000 }
gfCNCPoint5[19909] = {X 315.4331, Y 15.5947, Z -7.1667, A 0.000, B 0.000, C 0.000 }
gfCNCPoint5[19910] = {X 314.7895, Y 16.2730, Z -7.1667, A 0.000, B 0.000, C 0.000 }
gfCNCPoint5[19911] = {X 314.7890, Y 40.9133, Z -7.1667, A 0.000, B 0.000, C 0.000 }
gfCNCPoint5[19912] = {X 315.4271, Y 41.5843, Z -7.1667, A 0.000, B 0.000, C 0.000 }
gfCNCPoint5[19913] = {X 315.9076, Y 42.3758, Z -7.1667, A 0.000, B 0.000, C 0.000 }
gfCNCPoint5[19914] = {X 316.2083, Y 43.2516, Z -7.1667, A 0.000, B 0.000, C 0.000 }
gfCNCPoint5[19915] = {X 316.3156, Y 44.1713, Z -7.1667, A 0.000, B 0.000, C 0.000 }
gfCNCPoint5[19916] = {X 316.3157, Y 45.0000, Z -7.1667, A 0.000, B 0.000, C 0.000 }
gfCNCPoint5[19917] = {X 316.2074, Y 45.9613, Z -7.1667, A 0.000, B 0.000, C 0.000 }
gfCNCPoint5[19918] = {X 315.8879, Y 46.8744, Z -7.1667, A 0.000, B 0.000, C 0.000 }
gfCNCPoint5[19919] = {X 315.3732, Y 47.6935, Z -7.1667, A 0.000, B 0.000, C 0.000 }
gfCNCPoint5[19920] = {X 314.6892, Y 48.3775, Z -7.1667, A 0.000, B 0.000, C 0.000 }
gfCNCPoint5[19921] = {X 313.8701, Y 48.8922, Z -7.1667, A 0.000, B 0.000, C 0.000 }
gfCNCPoint5[19922] = {X 312.9570, Y 49.2117, Z -7.1667, A 0.000, B 0.000, C 0.000 }
gfCNCPoint5[19923] = {X 311.9957, Y 49.3200, Z -7.1667, A 0.000, B 0.000, C 0.000 }
gfCNCPoint5[19924] = {X 305.5523, Y 49.3200, Z -7.1667, A 0.000, B 0.000, C 0.000 }
gfCNCPoint5[19925] = {X 304.5958, Y 49.2128, Z -7.1667, A 0.000, B 0.000, C 0.000 }
gfCNCPoint5[19926] = {X 303.6868, Y 48.8965, Z -7.1667, A 0.000, B 0.000, C 0.000 }
gfCNCPoint5[19927] = {X 302.8704, Y 48.3868, Z -7.1667, A 0.000, B 0.000, C 0.000 }
gfCNCPoint5[19928] = {X 302.1872, Y 47.7090, Z -7.1667, A 0.000, B 0.000, C 0.000 }
gfCNCPoint5[19929] = {X 301.6709, Y 46.8967, Z -7.1667, A 0.000, B 0.000, C 0.000 }
gfCNCPoint5[19930] = {X 301.3473, Y 45.9903, Z -7.1667, A 0.000, B 0.000, C 0.000 }
gfCNCPoint5[19931] = {X 301.2324, Y 45.0348, Z -7.1667, A 0.000, B 0.000, C 0.000 }
gfCNCPoint5[19932] = {X 301.2323, Y 44.2014, Z -7.1667, A 0.000, B 0.000, C 0.000 }
gfCNCPoint5[19933] = {X 301.3495, Y 43.2653, Z -7.1667, A 0.000, B 0.000, C 0.000 }
gfCNCPoint5[19934] = {X 301.6523, Y 42.3718, Z -7.1667, A 0.000, B 0.000, C 0.000 }
gfCNCPoint5[19935] = {X 302.1285, Y 41.5574, Z -7.1667, A 0.000, B 0.000, C 0.000 }
gfCNCPoint5[19936] = {X 302.7587, Y 40.8553, Z -7.1667, A 0.000, B 0.000, C 0.000 }
gfCNCPoint5[19937] = {X 302.7587, Y 34.0343, Z -7.1667, A 0.000, B 0.000, C 0.000 }
gfCNCPoint5[19938] = {X 293.8552, Y 34.0343, Z -7.1667, A 0.000, B 0.000, C 0.000 }
gfCNCPoint5[19939] = {X 293.8546, Y 40.9019, Z -7.1667, A 0.000, B 0.000, C 0.000 }
gfCNCPoint5[19940] = {X 294.4938, Y 41.5860, Z -7.1667, A 0.000, B 0.000, C 0.000 }
gfCNCPoint5[19941] = {X 294.9743, Y 42.3895, Z -7.1667, A 0.000, B 0.000, C 0.000 }
gfCNCPoint5[19942] = {X 295.2746, Y 43.2762, Z -7.1667, A 0.000, B 0.000, C 0.000 }
gfCNCPoint5[19943] = {X 295.3811, Y 44.2064, Z -7.1667, A 0.000, B 0.000, C 0.000 }
gfCNCPoint5[19944] = {X 295.3811, Y 45.0000, Z -7.1667, A 0.000, B 0.000, C 0.000 }
gfCNCPoint5[19945] = {X 295.2728, Y 45.9613, Z -7.1667, A 0.000, B 0.000, C 0.000 }
gfCNCPoint5[19946] = {X 294.9533, Y 46.8744, Z -7.1667, A 0.000, B 0.000, C 0.000 }
gfCNCPoint5[19947] = {X 294.4386, Y 47.6935, Z -7.1667, A 0.000, B 0.000, C 0.000 }
gfCNCPoint5[19948] = {X 293.7546, Y 48.3775, Z -7.1667, A 0.000, B 0.000, C 0.000 }
gfCNCPoint5[19949] = {X 292.9355, Y 48.8922, Z -7.1667, A 0.000, B 0.000, C 0.000 }
gfCNCPoint5[19950] = {X 292.0224, Y 49.2117, Z -7.1667, A 0.000, B 0.000, C 0.000 }
gfCNCPoint5[19951] = {X 291.0611, Y 49.3200, Z -7.1667, A 0.000, B 0.000, C 0.000 }
gfCNCPoint5[19952] = {X 284.6177, Y 49.3200, Z -7.1667, A 0.000, B 0.000, C 0.000 }
gfCNCPoint5[19953] = {X 283.6613, Y 49.2128, Z -7.1667, A 0.000, B 0.000, C 0.000 }
gfCNCPoint5[19954] = {X 282.7524, Y 48.8965, Z -7.1667, A 0.000, B 0.000, C 0.000 }
gfCNCPoint5[19955] = {X 281.9360, Y 48.3869, Z -7.1667, A 0.000, B 0.000, C 0.000 }
gfCNCPoint5[19956] = {X 281.2527, Y 47.7092, Z -7.1667, A 0.000, B 0.000, C 0.000 }
gfCNCPoint5[19957] = {X 280.7365, Y 46.8970, Z -7.1667, A 0.000, B 0.000, C 0.000 }
gfCNCPoint5[19958] = {X 280.4128, Y 45.9907, Z -7.1667, A 0.000, B 0.000, C 0.000 }
gfCNCPoint5[19959] = {X 280.2978, Y 45.0352, Z -7.1667, A 0.000, B 0.000, C 0.000 }
gfCNCPoint5[19960] = {X 280.2977, Y 44.2074, Z -7.1667, A 0.000, B 0.000, C 0.000 }
gfCNCPoint5[19961] = {X 280.4019, Y 43.2782, Z -7.1667, A 0.000, B 0.000, C 0.000 }
gfCNCPoint5[19962] = {X 280.7017, Y 42.3925, Z -7.1667, A 0.000, B 0.000, C 0.000 }
gfCNCPoint5[19963] = {X 281.1832, Y 41.5910, Z -7.1667, A 0.000, B 0.000, C 0.000 }
gfCNCPoint5[19964] = {X 281.8244, Y 40.9104, Z -7.1667, A 0.000, B 0.000, C 0.000 }
gfCNCPoint5[19965] = {X 281.8244, Y 28.5919, Z -7.1667, A 0.000, B 0.000, C 0.000 }
gfCNCPoint5[19966] = {X 277.8244, Y 28.5919, Z -7.1667, A 0.000, B 0.000, C 0.000 }
gfCNCPoint5[19967] = {X 281.9044, Y 28.5919, Z -7.1667, A 0.000, B 0.000, C 0.000 }
gfCNCPoint5[19968] = {X 281.9043, Y 16.2361, Z -7.1667, A 0.000, B 0.000, C 0.000 }
gfCNCPoint5[19969] = {X 281.2666, Y 15.5757, Z -7.1667, A 0.000, B 0.000, C 0.000 }
gfCNCPoint5[19970] = {X 280.7860, Y 14.7935, Z -7.1667, A 0.000, B 0.000, C 0.000 }
gfCNCPoint5[19971] = {X 280.4850, Y 13.9262, Z -7.1667, A 0.000, B 0.000, C 0.000 }
gfCNCPoint5[19972] = {X 280.3778, Y 13.0144, Z -7.1667, A 0.000, B 0.000, C 0.000 }
gfCNCPoint5[19973] = {X 280.3777, Y 12.1868, Z -7.1667, A 0.000, B 0.000, C 0.000 }
gfCNCPoint5[19974] = {X 280.4840, Y 11.2433, Z -7.1667, A 0.000, B 0.000, C 0.000 }
gfCNCPoint5[19975] = {X 280.7976, Y 10.3472, Z -7.1667, A 0.000, B 0.000, C 0.000 }
gfCNCPoint5[19976] = {X 281.3027, Y 9.5432, Z -7.1667, A 0.000, B 0.000, C 0.000 }
gfCNCPoint5[19977] = {X 281.9741, Y 8.8719, Z -7.1667, A 0.000, B 0.000, C 0.000 }
gfCNCPoint5[19978] = {X 282.7780, Y 8.3667, Z -7.1667, A 0.000, B 0.000, C 0.000 }
gfCNCPoint5[19979] = {X 283.6742, Y 8.0531, Z -7.1667, A 0.000, B 0.000, C 0.000 }
gfCNCPoint5[19980] = {X 284.6177, Y 7.9468, Z -7.1667, A 0.000, B 0.000, C 0.000 }
gfCNCPoint5[19981] = {X 291.0611, Y 7.9468, Z -7.1667, A 0.000, B 0.000, C 0.000 }
gfCNCPoint5[19982] = {X 292.0046, Y 8.0531, Z -7.1667, A 0.000, B 0.000, C 0.000 }
gfCNCPoint5[19983] = {X 292.9008, Y 8.3667, Z -7.1667, A 0.000, B 0.000, C 0.000 }
gfCNCPoint5[19984] = {X 293.7047, Y 8.8718, Z -7.1667, A 0.000, B 0.000, C 0.000 }
gfCNCPoint5[19985] = {X 294.3761, Y 9.5432, Z -7.1667, A 0.000, B 0.000, C 0.000 }
gfCNCPoint5[19986] = {X 294.8812, Y 10.3471, Z -7.1667, A 0.000, B 0.000, C 0.000 }
gfCNCPoint5[19987] = {X 295.1948, Y 11.2433, Z -7.1667, A 0.000, B 0.000, C 0.000 }
gfCNCPoint5[19988] = {X 295.3011, Y 12.1868, Z -7.1667, A 0.000, B 0.000, C 0.000 }
gfCNCPoint5[19989] = {X 295.3011, Y 12.9782, Z -7.1667, A 0.000, B 0.000, C 0.000 }
gfCNCPoint5[19990] = {X 295.1997, Y 13.8996, Z -7.1667, A 0.000, B 0.000, C 0.000 }
gfCNCPoint5[19991] = {X 294.9004, Y 14.7769, Z -7.1667, A 0.000, B 0.000, C 0.000 }
gfCNCPoint5[19992] = {X 294.4177, Y 15.5682, Z -7.1667, A 0.000, B 0.000, C 0.000 }
gfCNCPoint5[19993] = {X 293.7745, Y 16.2357, Z -7.1667, A 0.000, B 0.000, C 0.000 }
gfCNCPoint5[19994] = {X 293.7754, Y 22.2765, Z -7.1667, A 0.000, B 0.000, C 0.000 }
gfCNCPoint5[19995] = {X 302.8384, Y 22.2765, Z -7.1667, A 0.000, B 0.000, C 0.000 }
gfCNCPoint5[19996] = {X 302.8435, Y 16.2400, Z -7.1667, A 0.000, B 0.000, C 0.000 }
gfCNCPoint5[19997] = {X 302.2042, Y 15.5796, Z -7.1667, A 0.000, B 0.000, C 0.000 }
gfCNCPoint5[19998] = {X 301.7222, Y 14.7969, Z -7.1667, A 0.000, B 0.000, C 0.000 }
gfCNCPoint5[19999] = {X 301.4202, Y 13.9287, Z -7.1667, A 0.000, B 0.000, C 0.000 }
gfCNCPoint5[20000] = {X 301.3124, Y 13.0158, Z -7.1667, A 0.000, B 0.000, C 0.000 }
gfCNCPoint5[20001] = {X 301.3123, Y 12.1868, Z -7.1667, A 0.000, B 0.000, C 0.000 }
gfCNCPoint5[20002] = {X 301.4186, Y 11.2433, Z -7.1667, A 0.000, B 0.000, C 0.000 }
gfCNCPoint5[20003] = {X 301.7321, Y 10.3471, Z -7.1667, A 0.000, B 0.000, C 0.000 }
gfCNCPoint5[20004] = {X 302.2373, Y 9.5432, Z -7.1667, A 0.000, B 0.000, C 0.000 }
gfCNCPoint5[20005] = {X 302.9087, Y 8.8718, Z -7.1667, A 0.000, B 0.000, C 0.000 }
gfCNCPoint5[20006] = {X 303.7126, Y 8.3667, Z -7.1667, A 0.000, B 0.000, C 0.000 }
gfCNCPoint5[20007] = {X 304.6088, Y 8.0531, Z -7.1667, A 0.000, B 0.000, C 0.000 }
gfCNCPoint5[20008] = {X 305.5523, Y 7.9468, Z -7.1667, A 0.000, B 0.000, C 0.000 }
gfCNCPoint5[20009] = {X 311.9957, Y 7.9468, Z -7.1667, A 0.000, B 0.000, C 0.000 }
gfCNCPoint5[20010] = {X 312.9392, Y 8.0531, Z -7.1667, A 0.000, B 0.000, C 0.000 }
gfCNCPoint5[20011] = {X 313.8354, Y 8.3667, Z -7.1667, A 0.000, B 0.000, C 0.000 }
gfCNCPoint5[20012] = {X 314.6393, Y 8.8718, Z -7.1667, A 0.000, B 0.000, C 0.000 }
gfCNCPoint5[20013] = {X 315.3107, Y 9.5432, Z -7.1667, A 0.000, B 0.000, C 0.000 }
gfCNCPoint5[20014] = {X 315.8158, Y 10.3471, Z -7.1667, A 0.000, B 0.000, C 0.000 }
gfCNCPoint5[20015] = {X 316.1294, Y 11.2433, Z -7.1667, A 0.000, B 0.000, C 0.000 }
gfCNCPoint5[20016] = {X 316.2357, Y 12.1868, Z -7.1667, A 0.000, B 0.000, C 0.000 }
gfCNCPoint5[20017] = {X 316.2357, Y 12.9782, Z -7.1667, A 0.000, B 0.000, C 0.000 }
gfCNCPoint5[20018] = {X 316.1344, Y 13.8995, Z -7.1667, A 0.000, B 0.000, C 0.000 }
gfCNCPoint5[20019] = {X 315.8352, Y 14.7769, Z -7.1667, A 0.000, B 0.000, C 0.000 }
gfCNCPoint5[20020] = {X 315.3526, Y 15.5682, Z -7.1667, A 0.000, B 0.000, C 0.000 }
gfCNCPoint5[20021] = {X 314.7095, Y 16.2358, Z -7.1667, A 0.000, B 0.000, C 0.000 }
gfCNCPoint5[20022] = {X 314.7090, Y 40.9514, Z -7.1667, A 0.000, B 0.000, C 0.000 }
gfCNCPoint5[20023] = {X 314.7373, Y 40.9744, Z -7.1667, A 0.000, B 0.000, C 0.000 }
gfCNCPoint5[20024] = {X 315.3636, Y 41.6329, Z -7.1667, A 0.000, B 0.000, C 0.000 }
gfCNCPoint5[20025] = {X 315.8351, Y 42.4098, Z -7.1667, A 0.000, B 0.000, C 0.000 }
gfCNCPoint5[20026] = {X 316.1303, Y 43.2693, Z -7.1667, A 0.000, B 0.000, C 0.000 }
gfCNCPoint5[20027] = {X 316.2356, Y 44.1720, Z -7.1667, A 0.000, B 0.000, C 0.000 }
gfCNCPoint5[20028] = {X 316.2357, Y 45.0000, Z -7.1667, A 0.000, B 0.000, C 0.000 }
gfCNCPoint5[20029] = {X 316.1294, Y 45.9435, Z -7.1667, A 0.000, B 0.000, C 0.000 }
gfCNCPoint5[20030] = {X 315.8158, Y 46.8397, Z -7.1667, A 0.000, B 0.000, C 0.000 }
gfCNCPoint5[20031] = {X 315.3107, Y 47.6436, Z -7.1667, A 0.000, B 0.000, C 0.000 }
gfCNCPoint5[20032] = {X 314.6393, Y 48.3150, Z -7.1667, A 0.000, B 0.000, C 0.000 }
gfCNCPoint5[20033] = {X 313.8354, Y 48.8201, Z -7.1667, A 0.000, B 0.000, C 0.000 }
gfCNCPoint5[20034] = {X 312.9392, Y 49.1337, Z -7.1667, A 0.000, B 0.000, C 0.000 }
gfCNCPoint5[20035] = {X 311.9957, Y 49.2400, Z -7.1667, A 0.000, B 0.000, C 0.000 }
gfCNCPoint5[20036] = {X 305.5523, Y 49.2400, Z -7.1667, A 0.000, B 0.000, C 0.000 }
gfCNCPoint5[20037] = {X 304.6135, Y 49.1348, Z -7.1667, A 0.000, B 0.000, C 0.000 }
gfCNCPoint5[20038] = {X 303.7214, Y 48.8243, Z -7.1667, A 0.000, B 0.000, C 0.000 }
gfCNCPoint5[20039] = {X 302.9201, Y 48.3241, Z -7.1667, A 0.000, B 0.000, C 0.000 }
gfCNCPoint5[20040] = {X 302.2495, Y 47.6588, Z -7.1667, A 0.000, B 0.000, C 0.000 }
gfCNCPoint5[20041] = {X 301.7428, Y 46.8616, Z -7.1667, A 0.000, B 0.000, C 0.000 }
gfCNCPoint5[20042] = {X 301.4252, Y 45.9720, Z -7.1667, A 0.000, B 0.000, C 0.000 }
gfCNCPoint5[20043] = {X 301.3124, Y 45.0341, Z -7.1667, A 0.000, B 0.000, C 0.000 }
gfCNCPoint5[20044] = {X 301.3123, Y 44.2033, Z -7.1667, A 0.000, B 0.000, C 0.000 }
gfCNCPoint5[20045] = {X 301.4294, Y 43.2746, Z -7.1667, A 0.000, B 0.000, C 0.000 }
gfCNCPoint5[20046] = {X 301.7324, Y 42.3890, Z -7.1667, A 0.000, B 0.000, C 0.000 }
gfCNCPoint5[20047] = {X 302.2088, Y 41.5832, Z -7.1667, A 0.000, B 0.000, C 0.000 }
gfCNCPoint5[20048] = {X 302.8387, Y 40.8909, Z -7.1667, A 0.000, B 0.000, C 0.000 }
gfCNCPoint5[20049] = {X 302.8387, Y 33.9543, Z -7.1667, A 0.000, B 0.000, C 0.000 }
gfCNCPoint5[20050] = {X 293.7752, Y 33.9543, Z -7.1667, A 0.000, B 0.000, C 0.000 }
gfCNCPoint5[20051] = {X 293.7746, Y 40.9387, Z -7.1667, A 0.000, B 0.000, C 0.000 }
gfCNCPoint5[20052] = {X 294.4134, Y 41.6123, Z -7.1667, A 0.000, B 0.000, C 0.000 }
gfCNCPoint5[20053] = {X 294.8940, Y 42.4065, Z -7.1667, A 0.000, B 0.000, C 0.000 }
gfCNCPoint5[20054] = {X 295.1945, Y 43.2848, Z -7.1667, A 0.000, B 0.000, C 0.000 }
gfCNCPoint5[20055] = {X 295.3011, Y 44.2070, Z -7.1667, A 0.000, B 0.000, C 0.000 }
gfCNCPoint5[20056] = {X 295.3011, Y 45.0000, Z -7.1667, A 0.000, B 0.000, C 0.000 }
gfCNCPoint5[20057] = {X 295.1948, Y 45.9435, Z -7.1667, A 0.000, B 0.000, C 0.000 }
gfCNCPoint5[20058] = {X 294.8812, Y 46.8397, Z -7.1667, A 0.000, B 0.000, C 0.000 }
gfCNCPoint5[20059] = {X 294.3761, Y 47.6436, Z -7.1667, A 0.000, B 0.000, C 0.000 }
gfCNCPoint5[20060] = {X 293.7047, Y 48.3150, Z -7.1667, A 0.000, B 0.000, C 0.000 }
gfCNCPoint5[20061] = {X 292.9008, Y 48.8201, Z -7.1667, A 0.000, B 0.000, C 0.000 }
gfCNCPoint5[20062] = {X 292.0046, Y 49.1337, Z -7.1667, A 0.000, B 0.000, C 0.000 }
gfCNCPoint5[20063] = {X 291.0611, Y 49.2400, Z -7.1667, A 0.000, B 0.000, C 0.000 }
gfCNCPoint5[20064] = {X 284.6177, Y 49.2400, Z -7.1667, A 0.000, B 0.000, C 0.000 }
gfCNCPoint5[20065] = {X 283.6790, Y 49.1348, Z -7.1667, A 0.000, B 0.000, C 0.000 }
gfCNCPoint5[20066] = {X 282.7869, Y 48.8244, Z -7.1667, A 0.000, B 0.000, C 0.000 }
gfCNCPoint5[20067] = {X 281.9857, Y 48.3242, Z -7.1667, A 0.000, B 0.000, C 0.000 }
gfCNCPoint5[20068] = {X 281.3150, Y 47.6590, Z -7.1667, A 0.000, B 0.000, C 0.000 }
gfCNCPoint5[20069] = {X 280.8083, Y 46.8619, Z -7.1667, A 0.000, B 0.000, C 0.000 }
gfCNCPoint5[20070] = {X 280.4907, Y 45.9723, Z -7.1667, A 0.000, B 0.000, C 0.000 }
gfCNCPoint5[20071] = {X 280.3778, Y 45.0345, Z -7.1667, A 0.000, B 0.000, C 0.000 }
gfCNCPoint5[20072] = {X 280.3777, Y 44.2078, Z -7.1667, A 0.000, B 0.000, C 0.000 }
gfCNCPoint5[20073] = {X 280.4820, Y 43.2866, Z -7.1667, A 0.000, B 0.000, C 0.000 }
gfCNCPoint5[20074] = {X 280.7820, Y 42.4095, Z -7.1667, A 0.000, B 0.000, C 0.000 }
gfCNCPoint5[20075] = {X 281.2637, Y 41.6174, Z -7.1667, A 0.000, B 0.000, C 0.000 }
gfCNCPoint5[20076] = {X 281.9044, Y 40.9475, Z -7.1667, A 0.000, B 0.000, C 0.000 }
gfCNCPoint5[20077] = {X 281.9044, Y 28.5919, Z -7.1667, A 0.000, B 0.000, C 0.000 }
gfCNCPoint5[20078] = {X 277.9044, Y 28.5919, Z -7.1667, A 0.000, B 0.000, C 0.000 }
gfCNCPoint5[20079] = {X 281.9844, Y 28.5919, Z -7.1667, A 0.000, B 0.000, C 0.000 }
gfCNCPoint5[20080] = {X 281.9843, Y 16.1984, Z -7.1667, A 0.000, B 0.000, C 0.000 }
gfCNCPoint5[20081] = {X 281.3471, Y 15.5488, Z -7.1667, A 0.000, B 0.000, C 0.000 }
gfCNCPoint5[20082] = {X 280.8663, Y 14.7761, Z -7.1667, A 0.000, B 0.000, C 0.000 }
gfCNCPoint5[20083] = {X 280.5651, Y 13.9174, Z -7.1667, A 0.000, B 0.000, C 0.000 }
gfCNCPoint5[20084] = {X 280.4578, Y 13.0137, Z -7.1667, A 0.000, B 0.000, C 0.000 }
gfCNCPoint5[20085] = {X 280.4577, Y 12.1868, Z -7.1667, A 0.000, B 0.000, C 0.000 }
gfCNCPoint5[20086] = {X 280.5620, Y 11.2611, Z -7.1667, A 0.000, B 0.000, C 0.000 }
gfCNCPoint5[20087] = {X 280.8696, Y 10.3819, Z -7.1667, A 0.000, B 0.000, C 0.000 }
gfCNCPoint5[20088] = {X 281.3652, Y 9.5931, Z -7.1667, A 0.000, B 0.000, C 0.000 }
gfCNCPoint5[20089] = {X 282.0240, Y 8.9344, Z -7.1667, A 0.000, B 0.000, C 0.000 }
gfCNCPoint5[20090] = {X 282.8127, Y 8.4388, Z -7.1667, A 0.000, B 0.000, C 0.000 }
gfCNCPoint5[20091] = {X 283.6920, Y 8.1311, Z -7.1667, A 0.000, B 0.000, C 0.000 }
gfCNCPoint5[20092] = {X 284.6177, Y 8.0268, Z -7.1667, A 0.000, B 0.000, C 0.000 }
gfCNCPoint5[20093] = {X 291.0611, Y 8.0268, Z -7.1667, A 0.000, B 0.000, C 0.000 }
gfCNCPoint5[20094] = {X 291.9868, Y 8.1311, Z -7.1667, A 0.000, B 0.000, C 0.000 }
gfCNCPoint5[20095] = {X 292.8661, Y 8.4388, Z -7.1667, A 0.000, B 0.000, C 0.000 }
gfCNCPoint5[20096] = {X 293.6549, Y 8.9344, Z -7.1667, A 0.000, B 0.000, C 0.000 }
gfCNCPoint5[20097] = {X 294.3136, Y 9.5931, Z -7.1667, A 0.000, B 0.000, C 0.000 }
gfCNCPoint5[20098] = {X 294.8092, Y 10.3819, Z -7.1667, A 0.000, B 0.000, C 0.000 }
gfCNCPoint5[20099] = {X 295.1168, Y 11.2611, Z -7.1667, A 0.000, B 0.000, C 0.000 }
gfCNCPoint5[20100] = {X 295.2211, Y 12.1868, Z -7.1667, A 0.000, B 0.000, C 0.000 }
gfCNCPoint5[20101] = {X 295.2211, Y 12.9782, Z -7.1667, A 0.000, B 0.000, C 0.000 }
gfCNCPoint5[20102] = {X 295.1255, Y 13.8649, Z -7.1667, A 0.000, B 0.000, C 0.000 }
gfCNCPoint5[20103] = {X 294.8431, Y 14.7108, Z -7.1667, A 0.000, B 0.000, C 0.000 }
gfCNCPoint5[20104] = {X 294.3868, Y 15.4771, Z -7.1667, A 0.000, B 0.000, C 0.000 }
gfCNCPoint5[20105] = {X 293.7778, Y 16.1285, Z -7.1667, A 0.000, B 0.000, C 0.000 }
gfCNCPoint5[20106] = {X 293.6945, Y 16.1985, Z -7.1667, A 0.000, B 0.000, C 0.000 }
gfCNCPoint5[20107] = {X 293.6954, Y 22.3565, Z -7.1667, A 0.000, B 0.000, C 0.000 }
gfCNCPoint5[20108] = {X 302.9183, Y 22.3565, Z -7.1667, A 0.000, B 0.000, C 0.000 }
gfCNCPoint5[20109] = {X 302.9236, Y 16.2022, Z -7.1667, A 0.000, B 0.000, C 0.000 }
gfCNCPoint5[20110] = {X 302.2847, Y 15.5526, Z -7.1667, A 0.000, B 0.000, C 0.000 }
gfCNCPoint5[20111] = {X 301.8025, Y 14.7794, Z -7.1667, A 0.000, B 0.000, C 0.000 }
gfCNCPoint5[20112] = {X 301.5003, Y 13.9199, Z -7.1667, A 0.000, B 0.000, C 0.000 }
gfCNCPoint5[20113] = {X 301.3924, Y 13.0151, Z -7.1667, A 0.000, B 0.000, C 0.000 }
gfCNCPoint5[20114] = {X 301.3923, Y 12.1868, Z -7.1667, A 0.000, B 0.000, C 0.000 }
gfCNCPoint5[20115] = {X 301.4966, Y 11.2611, Z -7.1667, A 0.000, B 0.000, C 0.000 }
gfCNCPoint5[20116] = {X 301.8042, Y 10.3819, Z -7.1667, A 0.000, B 0.000, C 0.000 }
gfCNCPoint5[20117] = {X 302.2998, Y 9.5931, Z -7.1667, A 0.000, B 0.000, C 0.000 }
gfCNCPoint5[20118] = {X 302.9585, Y 8.9344, Z -7.1667, A 0.000, B 0.000, C 0.000 }
gfCNCPoint5[20119] = {X 303.7473, Y 8.4388, Z -7.1667, A 0.000, B 0.000, C 0.000 }
gfCNCPoint5[20120] = {X 304.6266, Y 8.1311, Z -7.1667, A 0.000, B 0.000, C 0.000 }
gfCNCPoint5[20121] = {X 305.5523, Y 8.0268, Z -7.1667, A 0.000, B 0.000, C 0.000 }
gfCNCPoint5[20122] = {X 311.9957, Y 8.0268, Z -7.1667, A 0.000, B 0.000, C 0.000 }
gfCNCPoint5[20123] = {X 312.9214, Y 8.1311, Z -7.1667, A 0.000, B 0.000, C 0.000 }
gfCNCPoint5[20124] = {X 313.8007, Y 8.4388, Z -7.1667, A 0.000, B 0.000, C 0.000 }
gfCNCPoint5[20125] = {X 314.5894, Y 8.9344, Z -7.1667, A 0.000, B 0.000, C 0.000 }
gfCNCPoint5[20126] = {X 315.2481, Y 9.5931, Z -7.1667, A 0.000, B 0.000, C 0.000 }
gfCNCPoint5[20127] = {X 315.7438, Y 10.3819, Z -7.1667, A 0.000, B 0.000, C 0.000 }
gfCNCPoint5[20128] = {X 316.0514, Y 11.2611, Z -7.1667, A 0.000, B 0.000, C 0.000 }
gfCNCPoint5[20129] = {X 316.1557, Y 12.1868, Z -7.1667, A 0.000, B 0.000, C 0.000 }
gfCNCPoint5[20130] = {X 316.1557, Y 12.9782, Z -7.1667, A 0.000, B 0.000, C 0.000 }
gfCNCPoint5[20131] = {X 316.0542, Y 13.8913, Z -7.1667, A 0.000, B 0.000, C 0.000 }
gfCNCPoint5[20132] = {X 315.7548, Y 14.7598, Z -7.1667, A 0.000, B 0.000, C 0.000 }
gfCNCPoint5[20133] = {X 315.2721, Y 15.5414, Z -7.1667, A 0.000, B 0.000, C 0.000 }
gfCNCPoint5[20134] = {X 314.6295, Y 16.1981, Z -7.1667, A 0.000, B 0.000, C 0.000 }
gfCNCPoint5[20135] = {X 314.6290, Y 40.9896, Z -7.1667, A 0.000, B 0.000, C 0.000 }
gfCNCPoint5[20136] = {X 314.6839, Y 41.0340, Z -7.1667, A 0.000, B 0.000, C 0.000 }
gfCNCPoint5[20137] = {X 315.2990, Y 41.6802, Z -7.1667, A 0.000, B 0.000, C 0.000 }
gfCNCPoint5[20138] = {X 315.7622, Y 42.4427, Z -7.1667, A 0.000, B 0.000, C 0.000 }
gfCNCPoint5[20139] = {X 316.0522, Y 43.2865, Z -7.1667, A 0.000, B 0.000, C 0.000 }
gfCNCPoint5[20140] = {X 316.1556, Y 44.1727, Z -7.1667, A 0.000, B 0.000, C 0.000 }
gfCNCPoint5[20141] = {X 316.1557, Y 45.0000, Z -7.1667, A 0.000, B 0.000, C 0.000 }
gfCNCPoint5[20142] = {X 316.0514, Y 45.9257, Z -7.1667, A 0.000, B 0.000, C 0.000 }
gfCNCPoint5[20143] = {X 315.7438, Y 46.8050, Z -7.1667, A 0.000, B 0.000, C 0.000 }
gfCNCPoint5[20144] = {X 315.2481, Y 47.5937, Z -7.1667, A 0.000, B 0.000, C 0.000 }
gfCNCPoint5[20145] = {X 314.5894, Y 48.2524, Z -7.1667, A 0.000, B 0.000, C 0.000 }
gfCNCPoint5[20146] = {X 313.8007, Y 48.7480, Z -7.1667, A 0.000, B 0.000, C 0.000 }
gfCNCPoint5[20147] = {X 312.9214, Y 49.0557, Z -7.1667, A 0.000, B 0.000, C 0.000 }
gfCNCPoint5[20148] = {X 311.9957, Y 49.1600, Z -7.1667, A 0.000, B 0.000, C 0.000 }
gfCNCPoint5[20149] = {X 305.5523, Y 49.1600, Z -7.1667, A 0.000, B 0.000, C 0.000 }
gfCNCPoint5[20150] = {X 304.6312, Y 49.0568, Z -7.1667, A 0.000, B 0.000, C 0.000 }
gfCNCPoint5[20151] = {X 303.7559, Y 48.7522, Z -7.1667, A 0.000, B 0.000, C 0.000 }
gfCNCPoint5[20152] = {X 302.9698, Y 48.2613, Z -7.1667, A 0.000, B 0.000, C 0.000 }
gfCNCPoint5[20153] = {X 302.3118, Y 47.6087, Z -7.1667, A 0.000, B 0.000, C 0.000 }
gfCNCPoint5[20154] = {X 301.8147, Y 46.8265, Z -7.1667, A 0.000, B 0.000, C 0.000 }
gfCNCPoint5[20155] = {X 301.5030, Y 45.9537, Z -7.1667, A 0.000, B 0.000, C 0.000 }
gfCNCPoint5[20156] = {X 301.3924, Y 45.0335, Z -7.1667, A 0.000, B 0.000, C 0.000 }
gfCNCPoint5[20157] = {X 301.3923, Y 44.2051, Z -7.1667, A 0.000, B 0.000, C 0.000 }
gfCNCPoint5[20158] = {X 301.5094, Y 43.2840, Z -7.1667, A 0.000, B 0.000, C 0.000 }
gfCNCPoint5[20159] = {X 301.8126, Y 42.4063, Z -7.1667, A 0.000, B 0.000, C 0.000 }
gfCNCPoint5[20160] = {X 302.2891, Y 41.6093, Z -7.1667, A 0.000, B 0.000, C 0.000 }
gfCNCPoint5[20161] = {X 302.9187, Y 40.9268, Z -7.1667, A 0.000, B 0.000, C 0.000 }
gfCNCPoint5[20162] = {X 302.9187, Y 33.8743, Z -7.1667, A 0.000, B 0.000, C 0.000 }
gfCNCPoint5[20163] = {X 293.6952, Y 33.8743, Z -7.1667, A 0.000, B 0.000, C 0.000 }
gfCNCPoint5[20164] = {X 293.6946, Y 40.9759, Z -7.1667, A 0.000, B 0.000, C 0.000 }
gfCNCPoint5[20165] = {X 294.3329, Y 41.6389, Z -7.1667, A 0.000, B 0.000, C 0.000 }
gfCNCPoint5[20166] = {X 294.8137, Y 42.4237, Z -7.1667, A 0.000, B 0.000, C 0.000 }
gfCNCPoint5[20167] = {X 295.1145, Y 43.2935, Z -7.1667, A 0.000, B 0.000, C 0.000 }
gfCNCPoint5[20168] = {X 295.2211, Y 44.2076, Z -7.1667, A 0.000, B 0.000, C 0.000 }
gfCNCPoint5[20169] = {X 295.2211, Y 45.0000, Z -7.1667, A 0.000, B 0.000, C 0.000 }
gfCNCPoint5[20170] = {X 295.1168, Y 45.9257, Z -7.1667, A 0.000, B 0.000, C 0.000 }
gfCNCPoint5[20171] = {X 294.8092, Y 46.8050, Z -7.1667, A 0.000, B 0.000, C 0.000 }
gfCNCPoint5[20172] = {X 294.3136, Y 47.5937, Z -7.1667, A 0.000, B 0.000, C 0.000 }
gfCNCPoint5[20173] = {X 293.6549, Y 48.2524, Z -7.1667, A 0.000, B 0.000, C 0.000 }
gfCNCPoint5[20174] = {X 292.8661, Y 48.7480, Z -7.1667, A 0.000, B 0.000, C 0.000 }
gfCNCPoint5[20175] = {X 291.9868, Y 49.0557, Z -7.1667, A 0.000, B 0.000, C 0.000 }
gfCNCPoint5[20176] = {X 291.0611, Y 49.1600, Z -7.1667, A 0.000, B 0.000, C 0.000 }
gfCNCPoint5[20177] = {X 284.6177, Y 49.1600, Z -7.1667, A 0.000, B 0.000, C 0.000 }
gfCNCPoint5[20178] = {X 283.6967, Y 49.0568, Z -7.1667, A 0.000, B 0.000, C 0.000 }
gfCNCPoint5[20179] = {X 282.8214, Y 48.7522, Z -7.1667, A 0.000, B 0.000, C 0.000 }
gfCNCPoint5[20180] = {X 282.0353, Y 48.2615, Z -7.1667, A 0.000, B 0.000, C 0.000 }
gfCNCPoint5[20181] = {X 281.3774, Y 47.6088, Z -7.1667, A 0.000, B 0.000, C 0.000 }
gfCNCPoint5[20182] = {X 280.8802, Y 46.8267, Z -7.1667, A 0.000, B 0.000, C 0.000 }
gfCNCPoint5[20183] = {X 280.5685, Y 45.9540, Z -7.1667, A 0.000, B 0.000, C 0.000 }
gfCNCPoint5[20184] = {X 280.4578, Y 45.0339, Z -7.1667, A 0.000, B 0.000, C 0.000 }
gfCNCPoint5[20185] = {X 280.4577, Y 44.2081, Z -7.1667, A 0.000, B 0.000, C 0.000 }
gfCNCPoint5[20186] = {X 280.5621, Y 43.2951, Z -7.1667, A 0.000, B 0.000, C 0.000 }
gfCNCPoint5[20187] = {X 280.8624, Y 42.4266, Z -7.1667, A 0.000, B 0.000, C 0.000 }
gfCNCPoint5[20188] = {X 281.3441, Y 41.6441, Z -7.1667, A 0.000, B 0.000, C 0.000 }
gfCNCPoint5[20189] = {X 281.9844, Y 40.9849, Z -7.1667, A 0.000, B 0.000, C 0.000 }
gfCNCPoint5[20190] = {X 281.9844, Y 28.5919, Z -7.1667, A 0.000, B 0.000, C 0.000 }
gfCNCPoint5[20191] = {X 277.9844, Y 28.5919, Z -7.1667, A 0.000, B 0.000, C 0.000 }
gfCNCPoint5[20192] = {X 282.0644, Y 28.5919, Z -7.1667, A 0.000, B 0.000, C 0.000 }
gfCNCPoint5[20193] = {X 282.0643, Y 16.1603, Z -7.1667, A 0.000, B 0.000, C 0.000 }
gfCNCPoint5[20194] = {X 281.4275, Y 15.5215, Z -7.1667, A 0.000, B 0.000, C 0.000 }
gfCNCPoint5[20195] = {X 280.9467, Y 14.7585, Z -7.1667, A 0.000, B 0.000, C 0.000 }
gfCNCPoint5[20196] = {X 280.6452, Y 13.9085, Z -7.1667, A 0.000, B 0.000, C 0.000 }
gfCNCPoint5[20197] = {X 280.5378, Y 13.0130, Z -7.1667, A 0.000, B 0.000, C 0.000 }
gfCNCPoint5[20198] = {X 280.5377, Y 12.1868, Z -7.1667, A 0.000, B 0.000, C 0.000 }
gfCNCPoint5[20199] = {X 280.6400, Y 11.2789, Z -7.1667, A 0.000, B 0.000, C 0.000 }
gfCNCPoint5[20200] = {X 280.9417, Y 10.4166, Z -7.1667, A 0.000, B 0.000, C 0.000 }
gfCNCPoint5[20201] = {X 281.4278, Y 9.6430, Z -7.1667, A 0.000, B 0.000, C 0.000 }
gfCNCPoint5[20202] = {X 282.0738, Y 8.9969, Z -7.1667, A 0.000, B 0.000, C 0.000 }
gfCNCPoint5[20203] = {X 282.8474, Y 8.5109, Z -7.1667, A 0.000, B 0.000, C 0.000 }
gfCNCPoint5[20204] = {X 283.7098, Y 8.2091, Z -7.1667, A 0.000, B 0.000, C 0.000 }
gfCNCPoint5[20205] = {X 284.6177, Y 8.1068, Z -7.1667, A 0.000, B 0.000, C 0.000 }
gfCNCPoint5[20206] = {X 291.0611, Y 8.1068, Z -7.1667, A 0.000, B 0.000, C 0.000 }
gfCNCPoint5[20207] = {X 291.9690, Y 8.2091, Z -7.1667, A 0.000, B 0.000, C 0.000 }
gfCNCPoint5[20208] = {X 292.8314, Y 8.5109, Z -7.1667, A 0.000, B 0.000, C 0.000 }
gfCNCPoint5[20209] = {X 293.6050, Y 8.9969, Z -7.1667, A 0.000, B 0.000, C 0.000 }
gfCNCPoint5[20210] = {X 294.2510, Y 9.6430, Z -7.1667, A 0.000, B 0.000, C 0.000 }
gfCNCPoint5[20211] = {X 294.7371, Y 10.4166, Z -7.1667, A 0.000, B 0.000, C 0.000 }
gfCNCPoint5[20212] = {X 295.0388, Y 11.2789, Z -7.1667, A 0.000, B 0.000, C 0.000 }
gfCNCPoint5[20213] = {X 295.1411, Y 12.1868, Z -7.1667, A 0.000, B 0.000, C 0.000 }
gfCNCPoint5[20214] = {X 295.1411, Y 12.9782, Z -7.1667, A 0.000, B 0.000, C 0.000 }
gfCNCPoint5[20215] = {X 295.0473, Y 13.8478, Z -7.1667, A 0.000, B 0.000, C 0.000 }
gfCNCPoint5[20216] = {X 294.7704, Y 14.6775, Z -7.1667, A 0.000, B 0.000, C 0.000 }
gfCNCPoint5[20217] = {X 294.3229, Y 15.4290, Z -7.1667, A 0.000, B 0.000, C 0.000 }
gfCNCPoint5[20218] = {X 293.7255, Y 16.0679, Z -7.1667, A 0.000, B 0.000, C 0.000 }
gfCNCPoint5[20219] = {X 293.6679, Y 16.1166, Z -7.1667, A 0.000, B 0.000, C 0.000 }
gfCNCPoint5[20220] = {X 293.6095, Y 16.1643, Z -7.1667, A 0.000, B 0.000, C 0.000 }
gfCNCPoint5[20221] = {X 293.6145, Y 16.1985, Z -7.1667, A 0.000, B 0.000, C 0.000 }
gfCNCPoint5[20222] = {X 293.6155, Y 22.4365, Z -7.1667, A 0.000, B 0.000, C 0.000 }
gfCNCPoint5[20223] = {X 302.9982, Y 22.4365, Z -7.1667, A 0.000, B 0.000, C 0.000 }
gfCNCPoint5[20224] = {X 303.0036, Y 16.1640, Z -7.1667, A 0.000, B 0.000, C 0.000 }
gfCNCPoint5[20225] = {X 302.9451, Y 16.1164, Z -7.1667, A 0.000, B 0.000, C 0.000 }
gfCNCPoint5[20226] = {X 302.8875, Y 16.0676, Z -7.1667, A 0.000, B 0.000, C 0.000 }
gfCNCPoint5[20227] = {X 302.2957, Y 15.4360, Z -7.1667, A 0.000, B 0.000, C 0.000 }
gfCNCPoint5[20228] = {X 301.8505, Y 14.6937, Z -7.1667, A 0.000, B 0.000, C 0.000 }
gfCNCPoint5[20229] = {X 301.5719, Y 13.8742, Z -7.1667, A 0.000, B 0.000, C 0.000 }
gfCNCPoint5[20230] = {X 301.4724, Y 13.0144, Z -7.1667, A 0.000, B 0.000, C 0.000 }
gfCNCPoint5[20231] = {X 301.4723, Y 12.1868, Z -7.1667, A 0.000, B 0.000, C 0.000 }
gfCNCPoint5[20232] = {X 301.5745, Y 11.2789, Z -7.1667, A 0.000, B 0.000, C 0.000 }
gfCNCPoint5[20233] = {X 301.8763, Y 10.4166, Z -7.1667, A 0.000, B 0.000, C 0.000 }
gfCNCPoint5[20234] = {X 302.3624, Y 9.6430, Z -7.1667, A 0.000, B 0.000, C 0.000 }
gfCNCPoint5[20235] = {X 303.0084, Y 8.9969, Z -7.1667, A 0.000, B 0.000, C 0.000 }
gfCNCPoint5[20236] = {X 303.7820, Y 8.5109, Z -7.1667, A 0.000, B 0.000, C 0.000 }
gfCNCPoint5[20237] = {X 304.6444, Y 8.2091, Z -7.1667, A 0.000, B 0.000, C 0.000 }
gfCNCPoint5[20238] = {X 305.5523, Y 8.1068, Z -7.1667, A 0.000, B 0.000, C 0.000 }
gfCNCPoint5[20239] = {X 311.9957, Y 8.1068, Z -7.1667, A 0.000, B 0.000, C 0.000 }
gfCNCPoint5[20240] = {X 312.9036, Y 8.2091, Z -7.1667, A 0.000, B 0.000, C 0.000 }
gfCNCPoint5[20241] = {X 313.7660, Y 8.5109, Z -7.1667, A 0.000, B 0.000, C 0.000 }
gfCNCPoint5[20242] = {X 314.5396, Y 8.9969, Z -7.1667, A 0.000, B 0.000, C 0.000 }
gfCNCPoint5[20243] = {X 315.1856, Y 9.6430, Z -7.1667, A 0.000, B 0.000, C 0.000 }
gfCNCPoint5[20244] = {X 315.6717, Y 10.4166, Z -7.1667, A 0.000, B 0.000, C 0.000 }
gfCNCPoint5[20245] = {X 315.9734, Y 11.2789, Z -7.1667, A 0.000, B 0.000, C 0.000 }
gfCNCPoint5[20246] = {X 316.0757, Y 12.1868, Z -7.1667, A 0.000, B 0.000, C 0.000 }
gfCNCPoint5[20247] = {X 316.0757, Y 12.9782, Z -7.1667, A 0.000, B 0.000, C 0.000 }
gfCNCPoint5[20248] = {X 315.9741, Y 13.8829, Z -7.1667, A 0.000, B 0.000, C 0.000 }
gfCNCPoint5[20249] = {X 315.6744, Y 14.7426, Z -7.1667, A 0.000, B 0.000, C 0.000 }
gfCNCPoint5[20250] = {X 315.1915, Y 15.5144, Z -7.1667, A 0.000, B 0.000, C 0.000 }
gfCNCPoint5[20251] = {X 314.5495, Y 16.1599, Z -7.1667, A 0.000, B 0.000, C 0.000 }
gfCNCPoint5[20252] = {X 314.5490, Y 41.0278, Z -7.1667, A 0.000, B 0.000, C 0.000 }
gfCNCPoint5[20253] = {X 314.6336, Y 41.0962, Z -7.1667, A 0.000, B 0.000, C 0.000 }
gfCNCPoint5[20254] = {X 315.2363, Y 41.7299, Z -7.1667, A 0.000, B 0.000, C 0.000 }
gfCNCPoint5[20255] = {X 315.6902, Y 42.4775, Z -7.1667, A 0.000, B 0.000, C 0.000 }
gfCNCPoint5[20256] = {X 315.9743, Y 43.3047, Z -7.1667, A 0.000, B 0.000, C 0.000 }
gfCNCPoint5[20257] = {X 316.0756, Y 44.1734, Z -7.1667, A 0.000, B 0.000, C 0.000 }
gfCNCPoint5[20258] = {X 316.0757, Y 45.0000, Z -7.1667, A 0.000, B 0.000, C 0.000 }
gfCNCPoint5[20259] = {X 315.9734, Y 45.9079, Z -7.1667, A 0.000, B 0.000, C 0.000 }
gfCNCPoint5[20260] = {X 315.6717, Y 46.7702, Z -7.1667, A 0.000, B 0.000, C 0.000 }
gfCNCPoint5[20261] = {X 315.1856, Y 47.5438, Z -7.1667, A 0.000, B 0.000, C 0.000 }
gfCNCPoint5[20262] = {X 314.5396, Y 48.1899, Z -7.1667, A 0.000, B 0.000, C 0.000 }
gfCNCPoint5[20263] = {X 313.7660, Y 48.6760, Z -7.1667, A 0.000, B 0.000, C 0.000 }
gfCNCPoint5[20264] = {X 312.9036, Y 48.9777, Z -7.1667, A 0.000, B 0.000, C 0.000 }
gfCNCPoint5[20265] = {X 311.9957, Y 49.0800, Z -7.1667, A 0.000, B 0.000, C 0.000 }
gfCNCPoint5[20266] = {X 305.5523, Y 49.0800, Z -7.1667, A 0.000, B 0.000, C 0.000 }
gfCNCPoint5[20267] = {X 304.6489, Y 48.9787, Z -7.1667, A 0.000, B 0.000, C 0.000 }
gfCNCPoint5[20268] = {X 303.7905, Y 48.6800, Z -7.1667, A 0.000, B 0.000, C 0.000 }
gfCNCPoint5[20269] = {X 303.0194, Y 48.1986, Z -7.1667, A 0.000, B 0.000, C 0.000 }
gfCNCPoint5[20270] = {X 302.3741, Y 47.5585, Z -7.1667, A 0.000, B 0.000, C 0.000 }
gfCNCPoint5[20271] = {X 301.8865, Y 46.7914, Z -7.1667, A 0.000, B 0.000, C 0.000 }
gfCNCPoint5[20272] = {X 301.5809, Y 45.9353, Z -7.1667, A 0.000, B 0.000, C 0.000 }
gfCNCPoint5[20273] = {X 301.4724, Y 45.0328, Z -7.1667, A 0.000, B 0.000, C 0.000 }
gfCNCPoint5[20274] = {X 301.4723, Y 44.2070, Z -7.1667, A 0.000, B 0.000, C 0.000 }
gfCNCPoint5[20275] = {X 301.5893, Y 43.2934, Z -7.1667, A 0.000, B 0.000, C 0.000 }
gfCNCPoint5[20276] = {X 301.8927, Y 42.4238, Z -7.1667, A 0.000, B 0.000, C 0.000 }
gfCNCPoint5[20277] = {X 302.3694, Y 41.6357, Z -7.1667, A 0.000, B 0.000, C 0.000 }
gfCNCPoint5[20278] = {X 302.9987, Y 40.9632, Z -7.1667, A 0.000, B 0.000, C 0.000 }
gfCNCPoint5[20279] = {X 302.9987, Y 33.7943, Z -7.1667, A 0.000, B 0.000, C 0.000 }
gfCNCPoint5[20280] = {X 293.6152, Y 33.7943, Z -7.1667, A 0.000, B 0.000, C 0.000 }
gfCNCPoint5[20281] = {X 293.6146, Y 41.0135, Z -7.1667, A 0.000, B 0.000, C 0.000 }
gfCNCPoint5[20282] = {X 294.2524, Y 41.6657, Z -7.1667, A 0.000, B 0.000, C 0.000 }
gfCNCPoint5[20283] = {X 294.7334, Y 42.4410, Z -7.1667, A 0.000, B 0.000, C 0.000 }
gfCNCPoint5[20284] = {X 295.0344, Y 43.3022, Z -7.1667, A 0.000, B 0.000, C 0.000 }
gfCNCPoint5[20285] = {X 295.1411, Y 44.2082, Z -7.1667, A 0.000, B 0.000, C 0.000 }
gfCNCPoint5[20286] = {X 295.1411, Y 45.0000, Z -7.1667, A 0.000, B 0.000, C 0.000 }
gfCNCPoint5[20287] = {X 295.0388, Y 45.9079, Z -7.1667, A 0.000, B 0.000, C 0.000 }
gfCNCPoint5[20288] = {X 294.7371, Y 46.7702, Z -7.1667, A 0.000, B 0.000, C 0.000 }
gfCNCPoint5[20289] = {X 294.2510, Y 47.5438, Z -7.1667, A 0.000, B 0.000, C 0.000 }
gfCNCPoint5[20290] = {X 293.6050, Y 48.1899, Z -7.1667, A 0.000, B 0.000, C 0.000 }
gfCNCPoint5[20291] = {X 292.8314, Y 48.6760, Z -7.1667, A 0.000, B 0.000, C 0.000 }
gfCNCPoint5[20292] = {X 291.9690, Y 48.9777, Z -7.1667, A 0.000, B 0.000, C 0.000 }
gfCNCPoint5[20293] = {X 291.0611, Y 49.0800, Z -7.1667, A 0.000, B 0.000, C 0.000 }
gfCNCPoint5[20294] = {X 284.6177, Y 49.0800, Z -7.1667, A 0.000, B 0.000, C 0.000 }
gfCNCPoint5[20295] = {X 283.7144, Y 48.9788, Z -7.1667, A 0.000, B 0.000, C 0.000 }
gfCNCPoint5[20296] = {X 282.8560, Y 48.6801, Z -7.1667, A 0.000, B 0.000, C 0.000 }
gfCNCPoint5[20297] = {X 282.0850, Y 48.1987, Z -7.1667, A 0.000, B 0.000, C 0.000 }
gfCNCPoint5[20298] = {X 281.4397, Y 47.5587, Z -7.1667, A 0.000, B 0.000, C 0.000 }
gfCNCPoint5[20299] = {X 280.9521, Y 46.7916, Z -7.1667, A 0.000, B 0.000, C 0.000 }
gfCNCPoint5[20300] = {X 280.6464, Y 45.9356, Z -7.1667, A 0.000, B 0.000, C 0.000 }
gfCNCPoint5[20301] = {X 280.5378, Y 45.0332, Z -7.1667, A 0.000, B 0.000, C 0.000 }
gfCNCPoint5[20302] = {X 280.5377, Y 44.2085, Z -7.1667, A 0.000, B 0.000, C 0.000 }
gfCNCPoint5[20303] = {X 280.6422, Y 43.3037, Z -7.1667, A 0.000, B 0.000, C 0.000 }
gfCNCPoint5[20304] = {X 280.9427, Y 42.4439, Z -7.1667, A 0.000, B 0.000, C 0.000 }
gfCNCPoint5[20305] = {X 281.4247, Y 41.6711, Z -7.1667, A 0.000, B 0.000, C 0.000 }
gfCNCPoint5[20306] = {X 282.0644, Y 41.0228, Z -7.1667, A 0.000, B 0.000, C 0.000 }
gfCNCPoint5[20307] = {X 282.0644, Y 28.5919, Z -7.1667, A 0.000, B 0.000, C 0.000 }
gfCNCPoint5[20308] = {X 278.0644, Y 28.5919, Z -7.1667, A 0.000, B 0.000, C 0.000 }
gfCNCPoint5[20309] = {X 282.1444, Y 28.5919, Z -7.1667, A 0.000, B 0.000, C 0.000 }
gfCNCPoint5[20310] = {X 282.1443, Y 16.1216, Z -7.1667, A 0.000, B 0.000, C 0.000 }
gfCNCPoint5[20311] = {X 281.5026, Y 15.4873, Z -7.1667, A 0.000, B 0.000, C 0.000 }
gfCNCPoint5[20312] = {X 281.0195, Y 14.7253, Z -7.1667, A 0.000, B 0.000, C 0.000 }
gfCNCPoint5[20313] = {X 280.7194, Y 13.8745, Z -7.1667, A 0.000, B 0.000, C 0.000 }
gfCNCPoint5[20314] = {X 280.6177, Y 12.9780, Z -7.1667, A 0.000, B 0.000, C 0.000 }
gfCNCPoint5[20315] = {X 280.6177, Y 12.1868, Z -7.1667, A 0.000, B 0.000, C 0.000 }
gfCNCPoint5[20316] = {X 280.7180, Y 11.2967, Z -7.1667, A 0.000, B 0.000, C 0.000 }
gfCNCPoint5[20317] = {X 281.0138, Y 10.4513, Z -7.1667, A 0.000, B 0.000, C 0.000 }
gfCNCPoint5[20318] = {X 281.4903, Y 9.6929, Z -7.1667, A 0.000, B 0.000, C 0.000 }
gfCNCPoint5[20319] = {X 282.1237, Y 9.0595, Z -7.1667, A 0.000, B 0.000, C 0.000 }
gfCNCPoint5[20320] = {X 282.8821, Y 8.5829, Z -7.1667, A 0.000, B 0.000, C 0.000 }
gfCNCPoint5[20321] = {X 283.7276, Y 8.2871, Z -7.1667, A 0.000, B 0.000, C 0.000 }
gfCNCPoint5[20322] = {X 284.6177, Y 8.1868, Z -7.1667, A 0.000, B 0.000, C 0.000 }
gfCNCPoint5[20323] = {X 291.0611, Y 8.1868, Z -7.1667, A 0.000, B 0.000, C 0.000 }
gfCNCPoint5[20324] = {X 291.9512, Y 8.2871, Z -7.1667, A 0.000, B 0.000, C 0.000 }
gfCNCPoint5[20325] = {X 292.7967, Y 8.5829, Z -7.1667, A 0.000, B 0.000, C 0.000 }
gfCNCPoint5[20326] = {X 293.5551, Y 9.0595, Z -7.1667, A 0.000, B 0.000, C 0.000 }
gfCNCPoint5[20327] = {X 294.1885, Y 9.6929, Z -7.1667, A 0.000, B 0.000, C 0.000 }
gfCNCPoint5[20328] = {X 294.6650, Y 10.4513, Z -7.1667, A 0.000, B 0.000, C 0.000 }
gfCNCPoint5[20329] = {X 294.9608, Y 11.2967, Z -7.1667, A 0.000, B 0.000, C 0.000 }
gfCNCPoint5[20330] = {X 295.0611, Y 12.1868, Z -7.1667, A 0.000, B 0.000, C 0.000 }
gfCNCPoint5[20331] = {X 295.0609, Y 13.0192, Z -7.1667, A 0.000, B 0.000, C 0.000 }
gfCNCPoint5[20332] = {X 294.9625, Y 13.8608, Z -7.1667, A 0.000, B 0.000, C 0.000 }
gfCNCPoint5[20333] = {X 294.6890, Y 14.6628, Z -7.1667, A 0.000, B 0.000, C 0.000 }
gfCNCPoint5[20334] = {X 294.2528, Y 15.3892, Z -7.1667, A 0.000, B 0.000, C 0.000 }
gfCNCPoint5[20335] = {X 293.6733, Y 16.0073, Z -7.1667, A 0.000, B 0.000, C 0.000 }
gfCNCPoint5[20336] = {X 293.5963, Y 16.0721, Z -7.1667, A 0.000, B 0.000, C 0.000 }
gfCNCPoint5[20337] = {X 293.5177, Y 16.1348, Z -7.1667, A 0.000, B 0.000, C 0.000 }
gfCNCPoint5[20338] = {X 293.5345, Y 16.1928, Z -7.1667, A 0.000, B 0.000, C 0.000 }
gfCNCPoint5[20339] = {X 293.5355, Y 22.5165, Z -7.1667, A 0.000, B 0.000, C 0.000 }
gfCNCPoint5[20340] = {X 303.0782, Y 22.5165, Z -7.1667, A 0.000, B 0.000, C 0.000 }
gfCNCPoint5[20341] = {X 303.0785, Y 16.1929, Z -7.1667, A 0.000, B 0.000, C 0.000 }
gfCNCPoint5[20342] = {X 303.0955, Y 16.1346, Z -7.1667, A 0.000, B 0.000, C 0.000 }
gfCNCPoint5[20343] = {X 303.0168, Y 16.0718, Z -7.1667, A 0.000, B 0.000, C 0.000 }
gfCNCPoint5[20344] = {X 302.9398, Y 16.0070, Z -7.1667, A 0.000, B 0.000, C 0.000 }
gfCNCPoint5[20345] = {X 302.3542, Y 15.3806, Z -7.1667, A 0.000, B 0.000, C 0.000 }
gfCNCPoint5[20346] = {X 301.9156, Y 14.6438, Z -7.1667, A 0.000, B 0.000, C 0.000 }
gfCNCPoint5[20347] = {X 301.6441, Y 13.8305, Z -7.1667, A 0.000, B 0.000, C 0.000 }
gfCNCPoint5[20348] = {X 301.5523, Y 12.9780, Z -7.1667, A 0.000, B 0.000, C 0.000 }
gfCNCPoint5[20349] = {X 301.5523, Y 12.1868, Z -7.1667, A 0.000, B 0.000, C 0.000 }
gfCNCPoint5[20350] = {X 301.6525, Y 11.2967, Z -7.1667, A 0.000, B 0.000, C 0.000 }
gfCNCPoint5[20351] = {X 301.9484, Y 10.4513, Z -7.1667, A 0.000, B 0.000, C 0.000 }
gfCNCPoint5[20352] = {X 302.4249, Y 9.6929, Z -7.1667, A 0.000, B 0.000, C 0.000 }
gfCNCPoint5[20353] = {X 303.0583, Y 9.0595, Z -7.1667, A 0.000, B 0.000, C 0.000 }
gfCNCPoint5[20354] = {X 303.8167, Y 8.5829, Z -7.1667, A 0.000, B 0.000, C 0.000 }
gfCNCPoint5[20355] = {X 304.6622, Y 8.2871, Z -7.1667, A 0.000, B 0.000, C 0.000 }
gfCNCPoint5[20356] = {X 305.5523, Y 8.1868, Z -7.1667, A 0.000, B 0.000, C 0.000 }
gfCNCPoint5[20357] = {X 311.9957, Y 8.1868, Z -7.1667, A 0.000, B 0.000, C 0.000 }
gfCNCPoint5[20358] = {X 312.8858, Y 8.2871, Z -7.1667, A 0.000, B 0.000, C 0.000 }
gfCNCPoint5[20359] = {X 313.7313, Y 8.5829, Z -7.1667, A 0.000, B 0.000, C 0.000 }
gfCNCPoint5[20360] = {X 314.4897, Y 9.0595, Z -7.1667, A 0.000, B 0.000, C 0.000 }
gfCNCPoint5[20361] = {X 315.1230, Y 9.6929, Z -7.1667, A 0.000, B 0.000, C 0.000 }
gfCNCPoint5[20362] = {X 315.5996, Y 10.4513, Z -7.1667, A 0.000, B 0.000, C 0.000 }
gfCNCPoint5[20363] = {X 315.8954, Y 11.2967, Z -7.1667, A 0.000, B 0.000, C 0.000 }
gfCNCPoint5[20364] = {X 315.9957, Y 12.1868, Z -7.1667, A 0.000, B 0.000, C 0.000 }
gfCNCPoint5[20365] = {X 315.9955, Y 13.0192, Z -7.1667, A 0.000, B 0.000, C 0.000 }
gfCNCPoint5[20366] = {X 315.8870, Y 13.9044, Z -7.1667, A 0.000, B 0.000, C 0.000 }
gfCNCPoint5[20367] = {X 315.5850, Y 14.7436, Z -7.1667, A 0.000, B 0.000, C 0.000 }
gfCNCPoint5[20368] = {X 315.1045, Y 15.4950, Z -7.1667, A 0.000, B 0.000, C 0.000 }
gfCNCPoint5[20369] = {X 314.4695, Y 16.1213, Z -7.1667, A 0.000, B 0.000, C 0.000 }
gfCNCPoint5[20370] = {X 314.4690, Y 41.0660, Z -7.1667, A 0.000, B 0.000, C 0.000 }
gfCNCPoint5[20371] = {X 314.6078, Y 41.1794, Z -7.1667, A 0.000, B 0.000, C 0.000 }
gfCNCPoint5[20372] = {X 315.1935, Y 41.8059, Z -7.1667, A 0.000, B 0.000, C 0.000 }
gfCNCPoint5[20373] = {X 315.6322, Y 42.5427, Z -7.1667, A 0.000, B 0.000, C 0.000 }
gfCNCPoint5[20374] = {X 315.9038, Y 43.3562, Z -7.1667, A 0.000, B 0.000, C 0.000 }
gfCNCPoint5[20375] = {X 315.9957, Y 44.2089, Z -7.1667, A 0.000, B 0.000, C 0.000 }
gfCNCPoint5[20376] = {X 315.9957, Y 45.0000, Z -7.1667, A 0.000, B 0.000, C 0.000 }
gfCNCPoint5[20377] = {X 315.8954, Y 45.8901, Z -7.1667, A 0.000, B 0.000, C 0.000 }
gfCNCPoint5[20378] = {X 315.5996, Y 46.7355, Z -7.1667, A 0.000, B 0.000, C 0.000 }
gfCNCPoint5[20379] = {X 315.1230, Y 47.4940, Z -7.1667, A 0.000, B 0.000, C 0.000 }
gfCNCPoint5[20380] = {X 314.4897, Y 48.1273, Z -7.1667, A 0.000, B 0.000, C 0.000 }
gfCNCPoint5[20381] = {X 313.7313, Y 48.6039, Z -7.1667, A 0.000, B 0.000, C 0.000 }
gfCNCPoint5[20382] = {X 312.8858, Y 48.8997, Z -7.1667, A 0.000, B 0.000, C 0.000 }
gfCNCPoint5[20383] = {X 311.9957, Y 49.0000, Z -7.1667, A 0.000, B 0.000, C 0.000 }
gfCNCPoint5[20384] = {X 305.5523, Y 49.0000, Z -7.1667, A 0.000, B 0.000, C 0.000 }
gfCNCPoint5[20385] = {X 304.6622, Y 48.8997, Z -7.1667, A 0.000, B 0.000, C 0.000 }
gfCNCPoint5[20386] = {X 303.8167, Y 48.6039, Z -7.1667, A 0.000, B 0.000, C 0.000 }
gfCNCPoint5[20387] = {X 303.0583, Y 48.1273, Z -7.1667, A 0.000, B 0.000, C 0.000 }
gfCNCPoint5[20388] = {X 302.4249, Y 47.4939, Z -7.1667, A 0.000, B 0.000, C 0.000 }
gfCNCPoint5[20389] = {X 301.9484, Y 46.7355, Z -7.1667, A 0.000, B 0.000, C 0.000 }
gfCNCPoint5[20390] = {X 301.6525, Y 45.8901, Z -7.1667, A 0.000, B 0.000, C 0.000 }
gfCNCPoint5[20391] = {X 301.5523, Y 45.0000, Z -7.1667, A 0.000, B 0.000, C 0.000 }
gfCNCPoint5[20392] = {X 301.5523, Y 44.2088, Z -7.1667, A 0.000, B 0.000, C 0.000 }
gfCNCPoint5[20393] = {X 301.6693, Y 43.3029, Z -7.1667, A 0.000, B 0.000, C 0.000 }
gfCNCPoint5[20394] = {X 301.9729, Y 42.4414, Z -7.1667, A 0.000, B 0.000, C 0.000 }
gfCNCPoint5[20395] = {X 302.4497, Y 41.6623, Z -7.1667, A 0.000, B 0.000, C 0.000 }
gfCNCPoint5[20396] = {X 303.0787, Y 40.9999, Z -7.1667, A 0.000, B 0.000, C 0.000 }
gfCNCPoint5[20397] = {X 303.0787, Y 33.7143, Z -7.1667, A 0.000, B 0.000, C 0.000 }
gfCNCPoint5[20398] = {X 293.5352, Y 33.7143, Z -7.1667, A 0.000, B 0.000, C 0.000 }
gfCNCPoint5[20399] = {X 293.5346, Y 41.0516, Z -7.1667, A 0.000, B 0.000, C 0.000 }
gfCNCPoint5[20400] = {X 294.1720, Y 41.6929, Z -7.1667, A 0.000, B 0.000, C 0.000 }
gfCNCPoint5[20401] = {X 294.6530, Y 42.4585, Z -7.1667, A 0.000, B 0.000, C 0.000 }
gfCNCPoint5[20402] = {X 294.9543, Y 43.3110, Z -7.1667, A 0.000, B 0.000, C 0.000 }
gfCNCPoint5[20403] = {X 295.0611, Y 44.2089, Z -7.1667, A 0.000, B 0.000, C 0.000 }
gfCNCPoint5[20404] = {X 295.0611, Y 45.0000, Z -7.1667, A 0.000, B 0.000, C 0.000 }
gfCNCPoint5[20405] = {X 294.9608, Y 45.8901, Z -7.1667, A 0.000, B 0.000, C 0.000 }
gfCNCPoint5[20406] = {X 294.6650, Y 46.7355, Z -7.1667, A 0.000, B 0.000, C 0.000 }
gfCNCPoint5[20407] = {X 294.1885, Y 47.4940, Z -7.1667, A 0.000, B 0.000, C 0.000 }
gfCNCPoint5[20408] = {X 293.5551, Y 48.1273, Z -7.1667, A 0.000, B 0.000, C 0.000 }
gfCNCPoint5[20409] = {X 292.7967, Y 48.6039, Z -7.1667, A 0.000, B 0.000, C 0.000 }
gfCNCPoint5[20410] = {X 291.9512, Y 48.8997, Z -7.1667, A 0.000, B 0.000, C 0.000 }
gfCNCPoint5[20411] = {X 291.0611, Y 49.0000, Z -7.1667, A 0.000, B 0.000, C 0.000 }
gfCNCPoint5[20412] = {X 284.6177, Y 49.0000, Z -7.1667, A 0.000, B 0.000, C 0.000 }
gfCNCPoint5[20413] = {X 283.7276, Y 48.8997, Z -7.1667, A 0.000, B 0.000, C 0.000 }
gfCNCPoint5[20414] = {X 282.8821, Y 48.6039, Z -7.1667, A 0.000, B 0.000, C 0.000 }
gfCNCPoint5[20415] = {X 282.1237, Y 48.1273, Z -7.1667, A 0.000, B 0.000, C 0.000 }
gfCNCPoint5[20416] = {X 281.4903, Y 47.4939, Z -7.1667, A 0.000, B 0.000, C 0.000 }
gfCNCPoint5[20417] = {X 281.0138, Y 46.7355, Z -7.1667, A 0.000, B 0.000, C 0.000 }
gfCNCPoint5[20418] = {X 280.7180, Y 45.8901, Z -7.1667, A 0.000, B 0.000, C 0.000 }
gfCNCPoint5[20419] = {X 280.6177, Y 45.0000, Z -7.1667, A 0.000, B 0.000, C 0.000 }
gfCNCPoint5[20420] = {X 280.6177, Y 44.2088, Z -7.1667, A 0.000, B 0.000, C 0.000 }
gfCNCPoint5[20421] = {X 280.7223, Y 43.3124, Z -7.1667, A 0.000, B 0.000, C 0.000 }
gfCNCPoint5[20422] = {X 281.0231, Y 42.4614, Z -7.1667, A 0.000, B 0.000, C 0.000 }
